(* CODESYS project motor.library
   Company: ESO
   Description: Local Device Control - LDC Motor Library based on State Machine
   Version: 4.2.2.7
   Placeholder: ESO LDC Motor Library
   Author: Dan Popovic
   Title: ESO LDC Motor Library

Project tree, tasks and I/O mapping:
  libraries: Tc2_EtherCAT, * (Beckhoff Automation GmbH); Tc2_IoFunctions, * (Beckhoff Automation GmbH); Tc2_Math, * (Beckhoff Automation GmbH); Tc2_MC2, * (Beckhoff Automation GmbH); Tc2_MC2_Drive, * (Beckhoff Automation GmbH); Tc2_NC, * (Beckhoff Automation GmbH); Tc2_Standard, * (Beckhoff Automation GmbH); Tc2_System, * (Beckhoff Automation GmbH); Tc2_Utilities, * (Beckhoff Automation GmbH); Tc3_EventLogger, * (Beckhoff Automation GmbH); Tc3_Module, * (Beckhoff Automation GmbH); VisuDialogs, * (System); VisuSymbols, 3.5.10.0 (System)
  config/
    Mapping_with_new_EL6688_09_05.xml
    Mapping_with_old_EL6688_03_03.xml
    Mappings_SIM.xml
  00000000-0000-0000-0000-000000000000|config\Mapping_with_new_EL6688_09_05.xml
  00000000-0000-0000-0000-000000000000|config\Mapping_with_old_EL6688_03_03.xml
  00000000-0000-0000-0000-000000000000|config\Mappings_SIM.xml
  doc/
    AM8121_0F20_0000.xti
    EL7041_Phytron_57_500_1.2.xti
    EL7201_9014___AM8121_0F20_0000.xti
    MotorStateMachine.jpg
    Phytron_57_500_1.2_PID.xti
  00000000-0000-0000-0000-000000000000|doc\AM8121_0F20_0000.xti
  00000000-0000-0000-0000-000000000000|doc\EL7041_Phytron_57_500_1.2.xti
  00000000-0000-0000-0000-000000000000|doc\EL7201_9014___AM8121_0F20_0000.xti
  00000000-0000-0000-0000-000000000000|doc\MotorStateMachine.jpg
  00000000-0000-0000-0000-000000000000|doc\Phytron_57_500_1.2_PID.xti
  DUTs/
    Enumerated/
      Common/
        data type E_TIME_MODE
      Motor/
        data type E_DIRECTION
        data type E_MOTOR_AXIS_TYPE
        data type E_MOTOR_COMMAND
        data type E_MOTOR_ERROR
        data type E_MOTOR_EVENT
        data type E_MOTOR_INIT_ACTION
        data type E_MOTOR_INIT_SEQ_STATE
        data type E_MOTOR_INIT_STATE
        data type E_MOTOR_MODE
        data type E_MOTOR_MOVE_TYPE
        data type E_MOTOR_MOVING_STATE
        data type E_MOTOR_POST_INIT_STATE
        data type E_MOTOR_PRE_INIT_STATE
        data type E_MOTOR_RESET_STATE
        data type E_MOTOR_RPC_ERROR
        data type E_MOTOR_STATE
        data type E_MOTOR_STATUS
        data type E_MOTOR_SUBSTATE
        data type E_MOTOR_SWITCH_INDEX
      MultiAxis/
        data type E_MA_ADC_MOUNTING
        data type E_MA_AXES_ID
        data type E_MA_COMMAND
        data type E_MA_EVENT
        data type E_MA_MODE
        data type E_MA_ROTATOR_TYPE
        data type E_MA_RPC_ERROR
        data type E_MA_STATE
        data type E_MA_SUBSTATE
      Tracking/
        data type E_ADC_AXES_ID
        data type E_ADC_MODE
        data type E_DROT_MODE
        data type E_TRK_COMMAND
    Interfaces/
      interface ITrackCtrl: ComputeNextPos, HandleStates, Init, IsError, MoveInPos, MoveInSpeed, Reset
    Structures/
      Astro/
        data type T_ASTRO_ATMOSPHERE
        data type T_ASTRO_EL6688_DATA
        data type T_ASTRO_OUTPUT
        data type T_ASTRO_RA_DEC_RAD
        data type T_ASTRO_STAT
        data type T_ASTRO_TEL_DATA
        data type T_ASTRO_TEL_IF
        data type T_ASTRO_TRACKING_DATA
        data type T_ASTRO_UTC_TIME
        data type T_CPP_DEV_DATA
      CCS_Sim/
        data type T_CCS_CFG
        data type T_CCS_CTRL
        data type T_CCS_STAT
      Common/
        data type T_PTP_TIME
        data type T_TIMEVAL
        data type T_UTC_TIME
      Motor/
        data type T_MOTOR_ACTIVE_LOW
        data type T_MOTOR_AXIS_CFG
        data type T_MOTOR_CFG
        data type T_MOTOR_CTRL
        data type T_MOTOR_INFO
        data type T_MOTOR_INIT_STEP
        data type T_MOTOR_MC_PARAMETER
        data type T_MOTOR_MOTION
        data type T_MOTOR_SIGNAL
        data type T_MOTOR_SPEED
        data type T_MOTOR_STAT
        data type T_MOTOR_SWITCHES
        data type T_POSITION
      MultiAxis/
        data type T_MA_CFG
        data type T_MA_CTRL
        data type T_MA_SM_STAT
        data type T_MA_STAT
        data type T_MA_TOUT_CFG
      Simulation/
        data type T_SIM_MOTOR_CFG
        data type T_SIM_MOTOR_STAT
      Tracking/
        data type T_ADC_CFG
        data type T_ADC_CMD
        data type T_ADC_CTRL
        data type T_ADC_INFO
        data type T_ADC_STAT
        data type T_ADC_UNIT_CFG
        data type T_DROT_CFG
        data type T_DROT_CTRL
        data type T_DROT_INFO
        data type T_DROT_STAT
        data type T_TRK_CFG
        data type T_TRK_CTRL
        data type T_TRK_STAT
  GVLs/
    global variables GVL_TrkDefaultEnvironment
    global variables GVL_TrkSiteConstants
  lib/
  POUs/
    Astro/
      function block FB_ASTRO [ST]: M_Configure, M_CycleUpdate, M_DcAbsoluteTime, M_GetLeapSecond, M_TrkUpdate, M_Update
    CCS/
      function block FB_CCS_SIM [ST]: FB_init, GetParams, RPC_SetCoordinates, SetParams
    Functions/
      function F_astroDms2rad [ST]
      function F_astroHms2rad [ST]
      function F_astroRad2Hms [ST]
      function F_astroSplitHms [ST]
      function F_atan2 [ST]
      function F_DCTIME64_TO_ULINT [ST]
      function F_MOD [ST]
      function F_RAD2DMS_STRING [ST]
      function F_RAD2HMS_STRING [ST]
      function F_slaPa [ST]
      function F_timeGetAbsoluteDcTime [ST]
      function F_timeGetDcTime [ST]
      function F_timeGetUTC [ST]
      function F_timeUTCToJD [ST]
      function F_timeUTCToMJD [ST]
      function F_vltMod [ST]
      function F_vltSign [ST]
    Motor/
      function block FB_MOTOR [ST]: ActionClearNOVRAM, ActionErrExecute, ActionInitAbort, ActionInitComplete, ActionInitExecute, ActionInitReject, ActionMoveExecute, ActionResetExecute, ActionSetPosition, ActionStopExecute, ActionUnexpExecute, ActivityClearingNOVRAM, ActivityInitAborting, ActivityInitializing, ActivityMoving, ActivitySettingPosition, ActivityStopping, CheckForEvents, Dummy_UserExample, M_Configure, M_GetActualPos, M_GetOptimisedDistance, M_GetOptimisedPosition, M_GetRpcErrorText, M_HandleEnabled, M_MotorBrakeControl, M_MotorInitLock, M_MotorInitSeq, M_MotorPostInit, M_MotorPreInit, M_MotorReset, M_NormalizePos, M_NOVRAM_Clear, M_NOVRAM_Load, M_NOVRAM_Save, M_SetError, M_SetRpcStatus, M_UpdateSwitches, RPC_Disable, RPC_Enable, RPC_Init, RPC_MoveAbs, RPC_MoveRel, RPC_MoveVel, RPC_Reset, RPC_SetDebug, RPC_SetLog, RPC_Stop, UserPostInit, UserPostMove, UserPreInit, UserPreMove
      function block FB_MOTOR_BASE [ST]: ActionClearNOVRAM, ActionEnableExecute, ActionErrExecute, ActionInitAbort, ActionInitComplete, ActionInitExecute, ActionInitReject, ActionMoveExecute, ActionResetExecute, ActionSetPosition, ActionStopExecute, ActionUnexpExecute, ActivityClearingNOVRAM, ActivityInitAborting, ActivityInitializing, ActivityMoving, ActivitySettingPosition, ActivityStopping, CheckForEvents, M_GetErrorText, M_GetLogicalState, M_GetTimeInSec, M_LogEventDebug, M_LogEventEnd, M_LogEventError, M_LogEventGeneral, M_LogEventMoveAbs, M_LogEventMoveRel, M_LogEventMoveVel, M_LogEventStart, M_SetStatus, M_SetStatusDescription, ProcessEvents, SetAction, SetEvent, SetState, SetStatus
      function block FB_SIM_MOTOR [ST]: GetLogicalState, RPC_ResetConfig, RPC_SetCouplerState, RPC_SetDelay_Brake, RPC_SetDelay_SwitchActive, RPC_SetDelay_SwitchFind, RPC_SetFailure_BrakeFeedback
    MultiAxis/
      function block FB_MA_ADC [ST]: M_LogCommand, RPC_Disable, RPC_Enable, RPC_Init, RPC_MoveAbs, RPC_MoveAngle, RPC_MoveRel, RPC_MoveVel, RPC_Reset, RPC_StartTrack, RPC_Stop, RPC_StopTrack, User_ComputeAutoPos, User_ComputeNextPos, User_Configure, User_GetParams, User_SetParams
      function block FB_MA_BASE [ST]: ActionDisableExecute, ActionEnableExecute, ActionInitExecute, ActionMoveAbsExecute, ActionMoveVelExecute, ActionResetExecute, ActionStopExecute, ActionTrackExecute, ActivityDisabling, ActivityEnabling, ActivityInitialising, ActivityMoving, ActivityPresetting, ActivityResetting, ActivityStopping, ActivityTracking, CheckForEvents, M_AxesIdle, M_AxesInitialised, M_CheckAxesState, M_CheckError, M_Configure, M_GetMaxPosError, M_GetRpcErrorText, M_HomeMotors, M_LogCommand, M_LogEventGeneral, M_NextMove, M_NextMoveAbs, M_RestartTimer, M_SetInit, M_SetMode, M_SetRpcStatus, M_SetStatus, ProcessEvents, RPC_Init, SetAction, SetEvent, SetState, User_ComputeNextPos, User_Configure, User_GetParams, User_SetParams
      function block FB_MA_DROT [ST]: M_LogCommand, RPC_Disable, RPC_Enable, RPC_Init, RPC_MoveAbs, RPC_MoveAngle, RPC_MoveRel, RPC_MoveVel, RPC_Reset, RPC_StartTrack, RPC_Stop, RPC_StopTrack, User_ComputeNextPos, User_Configure, User_GetParams, User_SetParams
      function block FB_TRK_BASE [ST]: User_Configure, User_GetParams, User_SetParams
    program MAIN [ST]
  Version/
    global variables Global_Version
  VISUs/
    Motor/
      visualisation GUI_Motor001_Cfg
      visualisation GUI_Motor001_Ctrl
      visualisation GUI_Motor002_Cfg
      visualisation GUI_Motor002_Ctrl
    Templates/
      visualisation GUI_TEMPLATE_CCS_SIM
      visualisation GUI_TEMPLATE_MA_ADC
      visualisation GUI_TEMPLATE_MA_DROT
      visualisation GUI_TEMPLATE_MOTOR_CONFIG
      visualisation GUI_TEMPLATE_MOTOR_CONTROL
    Tracking/
      visualisation GUI_ADC_Motor1
      visualisation GUI_ADC_Motor2
      visualisation GUI_CCS_SIM
      visualisation GUI_DROT_Cfg
      visualisation GUI_DROT_Motor
      visualisation GUI_MA_ADC
      visualisation GUI_MA_DROT
  global variables GCL
  text list GlobalTextList
  global variables GPL
*)

// DUTs/Enumerated/Common/E_TIME_MODE
{attribute 'qualified_only'}
{attribute 'strict'}
TYPE E_TIME_MODE :
(
	LOCAL	:= 0,
	UTC		:= 1
);
END_TYPE

// DUTs/Enumerated/Motor/E_DIRECTION
{attribute 'qualified_only'}
{attribute 'strict'}
TYPE E_DIRECTION :
(
	NEGATIVE := 1,
	POSITIVE
);
END_TYPE

// DUTs/Enumerated/Motor/E_MOTOR_AXIS_TYPE
{attribute 'qualified_only'}
{attribute 'strict'}
TYPE E_MOTOR_AXIS_TYPE :
(
	LINEAR				:= 1,
	CIRCULAR,
	CIRCULAR_OPTIMISED
);
END_TYPE

// DUTs/Enumerated/Motor/E_MOTOR_COMMAND
{attribute 'qualified_only'}
{attribute 'strict'}
TYPE E_MOTOR_COMMAND :
(
	NONE	:= 0,
	
	// Commands corresponding to events - MUST match E_MOTOR_EVENT !!!
	RESET,
	INIT,
	STOP,
	ENABLE,
	DISABLE,
	MOTOR_MOVE,
	SET_POSITION,
	CLEAR_NOVRAM
);
END_TYPE

// DUTs/Enumerated/Motor/E_MOTOR_ERROR
{attribute 'qualified_only'}
// 'strict' cannot be used since we mix our own codes with TC codes
//{attribute 'strict'}
TYPE E_MOTOR_ERROR :
(
	OK					:= 0,
	HW_NOT_OP,			
	LOCAL,			
	INIT_ABORTED,		
	TIMEOUT_INIT,
	TIMEOUT_MOVE,
	TIMEOUT_RESET,
	TIMEOUT_SETPOS,
	TIMEOUT_USER_PREINIT,
	TIMEOUT_USER_POSTINIT,
	TIMEOUT_USER_PREMOVE,
	TIMEOUT_USER_POSTMOVE,
	SETPOS,
	STOP,
	
	ABORT,
	SW_LIMIT_LOWER,
	SW_LIMIT_UPPER,
	BRAKE_ACTIVE,
	BRAKE_ENGAGE,
	BRAKE_DISENGAGE,
	SWITCH_NOT_USED,
	ENABLE,
	NOVRAM_READ,
	NOVRAM_WRITE,
	SWITCH_EXIT,
	STOP_LIMITS_BOTH,
	HW_LIMITS_BOTH,
	IN_POS,
	LOCKED,
	SoE_ADS_ERROR,
	SoE_SERCOS_ERROR,

	// Simulator errors
	SIM_NOT_INITIALISED			:= 90,
	SIM_NULL_POINTER			:= 100,	

	// TwinCAT errors
	TC_VEL						:= 16929,	
	TC_NOT_READY_FOR_START		:= 16933,	
	TC_DISABLED_MOVE			:= 16992,	
	TC_BISECTION				:= 17022,	
	TC_MODULO_POS				:= 17026,	
	TC_STOP_ACTIVE				:= 17135,	
	TC_VEL_NEG					:= 17241,	
	TC_TARGET_LSW				:= 17504,	
	TC_TARGET_USW				:= 17505,	
	TC_FOLLOWING_ERROR			:= 17744,	
	TC_NOT_READY				:= 18000,	
	TC_IN_POS_6_SEC				:= 19207	

);
END_TYPE

// DUTs/Enumerated/Motor/E_MOTOR_EVENT
{attribute 'qualified_only'}
{attribute 'strict'}
TYPE E_MOTOR_EVENT :
(
	NONE	:= 0,
	
	(* events corresponding to commands - MUST match E_MOTOR_COMMAND *)
	RESET,
	INIT,
	STOP,
	ENABLE,
	DISABLE,
	MOTOR_MOVE,
	SET_POSITION,
	CLEAR_NOVRAM,
	
	(* 
		Events corresponding to internal events 
	*)
	
	MOVEDONE,		// Needed for detection of HW failures during initialisation
	STOPDONE,
	ENABLEDONE,
	DISABLEDONE,
	INITDONE,
	SETPOSDONE,
	

	HWOK,
	ERRLOCAL,
	ERRHW,
	ERRRESET,
	ERRFAULT,
	ERRINIT,
	ERRSTOP,
	ERRENABLE,
	ERRDISABLE,
	ERRBRAKE,
	ERRINPOS,
	ERRLOCKED,
	ERRTARGETPAR,
	ERRUSERPREINIT,
	ERRUSERPREMOVE,
	ERRUSERPOSTINIT,
	ERRUSERPOSTMOVE,
	TIMEOUT_MOVE,
	TIMEOUT_SETPOS,
	SW_LIMIT_LOWER,
	SW_LIMIT_UPPER
	
);
END_TYPE

// DUTs/Enumerated/Motor/E_MOTOR_INIT_ACTION
TYPE E_MOTOR_INIT_ACTION :
(
	MOTOR_INIT_ACTION_END				:= 0,
	MOTOR_INIT_ACTION_FIND_INDEX,
	MOTOR_INIT_ACTION_FIND_REF_LE,
	MOTOR_INIT_ACTION_FIND_REF_UE,
	MOTOR_INIT_ACTION_FIND_LHW,
	MOTOR_INIT_ACTION_FIND_UHW,
	MOTOR_INIT_ACTION_DELAY,
	MOTOR_INIT_ACTION_MOVE_ABS,
	MOTOR_INIT_ACTION_MOVE_REL,
	MOTOR_INIT_ACTION_CALIB_ABS,
	MOTOR_INIT_ACTION_CALIB_REL,
	MOTOR_INIT_ACTION_CALIB_SWITCH,
	// The following steps cannot be configured in the INIT sequence
	MOTOR_INIT_ACTION_STEP1_START,
	MOTOR_INIT_ACTION_STEP1_EXECUTE,
	MOTOR_INIT_ACTION_STEP2_START,
	MOTOR_INIT_ACTION_STEP2_EXECUTE,
	MOTOR_INIT_ACTION_STOP
);
END_TYPE

// DUTs/Enumerated/Motor/E_MOTOR_INIT_SEQ_STATE
TYPE E_MOTOR_INIT_SEQ_STATE :
(
	MOTOR_INIT_SEQ_STATE_START				:= 0,
	MOTOR_INIT_SEQ_STATE_EXECUTE,
	MOTOR_INIT_SEQ_STATE_END
);
END_TYPE

// DUTs/Enumerated/Motor/E_MOTOR_INIT_STATE
TYPE E_MOTOR_INIT_STATE :
(
	MOTOR_INIT_STATE_START				:= 0,
	MOTOR_INIT_STATE_RESET,
	MOTOR_INIT_STATE_WAIT_READY,
	MOTOR_INIT_STATE_PRE_INIT,
	MOTOR_INIT_STATE_USER_PRE_INIT,
	MOTOR_INIT_STATE_INIT_SEQ,
	MOTOR_INIT_STATE_INIT_LOCK,
	MOTOR_INIT_STATE_POST_INIT,
	MOTOR_INIT_STATE_USER_POST_INIT,
	MOTOR_INIT_STATE_SAVE_NOVRAM,
	MOTOR_INIT_STATE_END
);
END_TYPE

// DUTs/Enumerated/Motor/E_MOTOR_MODE
{attribute 'qualified_only'}
{attribute 'strict'}
TYPE E_MOTOR_MODE :
(
	POS				:= 0,
	VEL
);
END_TYPE

// DUTs/Enumerated/Motor/E_MOTOR_MOVE_TYPE
{attribute 'qualified_only'}
{attribute 'strict'}
TYPE E_MOTOR_MOVE_TYPE :
(
	NONE	:= 0,
	
	ABSOLUTE,
	RELATIVE,
	VELOCITY,
	TRACKING

);
END_TYPE

// DUTs/Enumerated/Motor/E_MOTOR_MOVING_STATE
TYPE E_MOTOR_MOVING_STATE :
(
	MOTOR_MOVING_STATE_NONE	:= 0,
	MOTOR_MOVING_STATE_ENABLE,
	MOTOR_MOVING_STATE_WAIT_BRAKES,
	MOTOR_MOVING_STATE_USER_PRE_MOVE,
	MOTOR_MOVING_STATE_WAIT_ABSOLUTE,
	MOTOR_MOVING_STATE_WAIT_OPTIMISED,
	MOTOR_MOVING_STATE_WAIT_VELOCITY,
	MOTOR_MOVING_STATE_USER_POST_MOVE,
	MOTOR_MOVING_STATE_APPLY_BRAKES,
	MOTOR_MOVING_STATE_DISABLE,
	MOTOR_MOVING_STATE_CHECK_IN_POS,
	MOTOR_MOVING_STATE_END
);
END_TYPE

// DUTs/Enumerated/Motor/E_MOTOR_POST_INIT_STATE
TYPE E_MOTOR_POST_INIT_STATE :
(
	MOTOR_POST_INIT_STATE_START	:= 0,
	MOTOR_POST_INIT_STATE_WRITE,
	MOTOR_POST_INIT_STATE_END
);
END_TYPE

// DUTs/Enumerated/Motor/E_MOTOR_PRE_INIT_STATE
TYPE E_MOTOR_PRE_INIT_STATE :
(
	MOTOR_PRE_INIT_STATE_START	:= 0,
	MOTOR_PRE_INIT_STATE_READ,
	MOTOR_PRE_INIT_STATE_GET_USER_UNITS,
	MOTOR_PRE_INIT_STATE_WRITE,
	MOTOR_PRE_INIT_STATE_END
);
END_TYPE

// DUTs/Enumerated/Motor/E_MOTOR_RESET_STATE
TYPE E_MOTOR_RESET_STATE :
(
	MOTOR_RESET_STATE_START	:= 0,
	MOTOR_RESET_STATE_SoE_RESET,
	MOTOR_RESET_STATE_SoE_WAIT_RESET,
	MOTOR_RESET_STATE_RESET_AXIS,
	MOTOR_RESET_STATE_WAIT,
	MOTOR_RESET_STATE_END
);
END_TYPE

// DUTs/Enumerated/Motor/E_MOTOR_RPC_ERROR
{attribute 'qualified_only'}
{attribute 'strict'}
TYPE E_MOTOR_RPC_ERROR :
(
	OK						:= 0,
	NOT_OP					:= -1,			
	NOT_NOTOP_READY			:= -2,			
	NOT_NOTOP_NOTREADY		:= -3,			
	LOCAL					:= -4,			
	SW_LIMIT_LOWER			:= -5,			
	SW_LIMIT_UPPER			:= -6,			
	INIT_WHILE_MOVING		:= -7,
	VEL_ZERO				:= -8,			
	VEL_NEG					:= -9,			
	VEL_MAX					:= -10			
);
END_TYPE

// DUTs/Enumerated/Motor/E_MOTOR_STATE
{attribute 'qualified_only'}
{attribute 'strict'}
TYPE E_MOTOR_STATE :
(
	NONE	:= 0,
	NOTOP,
	OP
);
END_TYPE

// DUTs/Enumerated/Motor/E_MOTOR_STATUS
{attribute 'qualified_only'}
{attribute 'strict'}
TYPE E_MOTOR_STATUS :
(
	OK	:= 0,
	ERROR,
	
	STANDING,
	MOVING

);
END_TYPE

// DUTs/Enumerated/Motor/E_MOTOR_SUBSTATE
{attribute 'qualified_only'}
{attribute 'strict'}
TYPE E_MOTOR_SUBSTATE :
(
	NONE					:= 0,
	
	NOTOP_NOTREADY			:= 100,
	NOTOP_READY				:= 101,
	NOTOP_INITIALIZING		:= 102,
	NOTOP_ABORTING			:= 107,
	NOTOP_CLEARING_NOVRAM	:= 108,
	
	NOTOP_ERROR				:= 199,
	
	
	OP_STANDSTILL			:= 216,            
	OP_MOVING				:= 217,
	OP_SETTING_POS			:= 218,
	OP_STOPPING				:= 219,
	
	OP_ERROR				:= 299
);
END_TYPE

// DUTs/Enumerated/Motor/E_MOTOR_SWITCH_INDEX
{attribute 'qualified_only'}
{attribute 'strict'}
TYPE E_MOTOR_SWITCH_INDEX :
(
	LSTOP	:= 0,
	LHW		:= 1,
	REF		:= 2,
	INDEX	:= 3,
	UHW		:= 4,
	USTOP	:= 5
);
END_TYPE

// DUTs/Enumerated/MultiAxis/E_MA_ADC_MOUNTING
TYPE E_MA_ADC_MOUNTING :
(
	// ADC positions should be the same due to oposite mounting of ADC units,
	// i.e. ADC2 = ADC1
	MA_ADC_MOUNTING_OPOSITE_SIDE := 0,
	// ADC positions should have oposite vales due to the same mounting of both ADC units,
	// i.e. ADC2 = -ADC1
	MA_ADC_MOUNTING_SAME_SIDE := 1
);
END_TYPE

// DUTs/Enumerated/MultiAxis/E_MA_AXES_ID
{attribute 'qualified_only'}
{attribute 'strict'}
TYPE E_MA_AXES_ID :
(
	ALL_AXES := 0,
	AXIS_1,
	AXIS_2,
	AXIS_3,
	AXIS_4,
	AXIS_5,
	AXIS_6
);
END_TYPE

// DUTs/Enumerated/MultiAxis/E_MA_COMMAND
{attribute 'qualified_only'}
{attribute 'strict'}
TYPE E_MA_COMMAND :
(
	NONE	:= 0,
	
	// Commands corresponding to events - MUST match E_MA_EVENT !!!
	RESET,
	INIT,
	STOP,
	ENABLE,
	DISABLE,
	MA_MOVE,
	START_TRACK,
	STOP_TRACK
);
END_TYPE

// DUTs/Enumerated/MultiAxis/E_MA_EVENT
{attribute 'qualified_only'}
{attribute 'strict'}
TYPE E_MA_EVENT :
(
	NONE	:= 0,
	
	(* events corresponding to commands - MUST match E_MA_COMMAND *)
	RESET,
	INIT,
	STOP,
	ENABLE,
	DISABLE,
	MA_MOVE,
	START_TRACK,
	STOP_TRACK,
	
	(* 
		Events corresponding to internal events 
	*)
	
	MOVEDONE,		// Needed for detection of HW failures during initialisation
	STOPDONE,
	ENABLEDONE,
	DISABLEDONE,
	INITDONE,
	TRACKDONE,
	TRACKEXIT,		// EICSSW-706: Tracking error >=  cfg.lrTrkThreshold => PRESETTING
	PRESETDONE,		// EICSSW-706: Presetting error < cfg.lrTrkThreshold => TRACKING
	

	HWOK,
	ERRLOCAL,
	ERRHW
	
);
END_TYPE

// DUTs/Enumerated/MultiAxis/E_MA_MODE
TYPE E_MA_MODE :
(
	// WARNING: modes shall be a positive number
	MA_MODE_ENG	:= 0
);
END_TYPE

// DUTs/Enumerated/MultiAxis/E_MA_ROTATOR_TYPE
{attribute 'qualified_only'}
{attribute 'strict'}
TYPE E_MA_ROTATOR_TYPE :
(
	DROT 	:= 0,	// Derotator
	ADAPTER := 1,	// Adapter
	ROTATOR := 2	// Rotator
);
END_TYPE

// DUTs/Enumerated/MultiAxis/E_MA_RPC_ERROR
{attribute 'qualified_only'}
{attribute 'strict'}
TYPE E_MA_RPC_ERROR :
(
	OK						:=  0,
	NOT_OP					:= -1,			
	NOT_NOTOP_READY	    	:= -2,			
	NOT_NOTOP_NOTREADY		:= -3,			
	LOCAL					:= -4,			
	SW_LIMIT_LOWER			:= -5,			
	SW_LIMIT_UPPER			:= -6,			
	INIT_WHILE_MOVING		:= -7,
	VEL_ZERO				:= -8,			
	VEL_NEG					:= -9,			
	VEL_MAX					:= -10			
);
END_TYPE

// DUTs/Enumerated/MultiAxis/E_MA_STATE
{attribute 'qualified_only'}
//{attribute 'strict'}
TYPE E_MA_STATE :
(
	NONE	:= 0,
	NOTOP,
	OP
);
END_TYPE

// DUTs/Enumerated/MultiAxis/E_MA_SUBSTATE
{attribute 'qualified_only'}
//{attribute 'strict'}
TYPE E_MA_SUBSTATE :
(
	NONE				:=   0,
	
	NOTOP_NOTREADY		:= 100,
	NOTOP_READY			:= 101,
	NOTOP_INITIALISING	:= 102,
	NOTOP_ABORTING		:= 107,
	
	NOTOP_RESETTING		:= 109,
	NOTOP_ENABLING		:= 110,

	NOTOP_ERROR			:= 199,

	
	OP_DISABLING 		:= 205,
	OP_STANDSTILL		:= 216,            
	OP_MOVING			:= 217,
	OP_SETTING_POS		:= 218,
	OP_STOPPING			:= 219,
	OP_TRACKING			:= 220,
	OP_PRESETTING		:= 221,

	OP_ERROR			:= 299

);
END_TYPE

// DUTs/Enumerated/Tracking/E_ADC_AXES_ID
{attribute 'qualified_only'}
{attribute 'strict'}
TYPE E_ADC_AXES_ID :
(
	ALL_AXES := 0,
	ADC_1,
	ADC_2
);
END_TYPE

// DUTs/Enumerated/Tracking/E_ADC_MODE
{attribute 'qualified_only'}
{attribute 'strict'}
TYPE E_ADC_MODE :
(
	// WARNING: modes shall be a positive number
	ENG   := 0, 
	OFF   := 1,
	AUTO  := 2
);
END_TYPE

// DUTs/Enumerated/Tracking/E_DROT_MODE
{attribute 'qualified_only'}
{attribute 'strict'}
TYPE E_DROT_MODE :
(
	ENG		:= 0,
	STAT	:= 1,
	SKY		:= 2,
	ELEV	:= 3,
	USER	:= 4
);
END_TYPE

// DUTs/Enumerated/Tracking/E_TRK_COMMAND
{attribute 'qualified_only'}
{attribute 'strict'}
TYPE E_TRK_COMMAND :
(
	NONE			:= 0,
	INIT			:= 1,
	STOP, 
	TRK_MOVE,
	START_TRACK,
	STOP_TRACK,
	RESET,
	ENABLE,
	DISABLE,
	MOVE_MASTER
);
END_TYPE

// DUTs/Structures/Astro/T_ASTRO_ATMOSPHERE
// Structure containing atmospheric conditions.
// To be updated by the WS driver, i.e. "scanning" from TEL
TYPE T_ASTRO_ATMOSPHERE :
STRUCT
	lrTemperature:	LREAL   := 12.0;	// Air temperature [degC]
	lrPressure:		LREAL   := 743.0;	// Atmospheric Pressure [mbar]
	lrHumidity:		LREAL   := 0.2;		// Relative humidity [0.0..1.0]
END_STRUCT
END_TYPE

// DUTs/Structures/Astro/T_ASTRO_EL6688_DATA
TYPE T_ASTRO_EL6688_DATA :
STRUCT
	Control_value_update_toggle:	BOOL;
	External_device_not_connected:	BOOL;
	Internal_time_stamp:			ULINT;
	External_time_stamp:			ULINT;
END_STRUCT
END_TYPE

// DUTs/Structures/Astro/T_ASTRO_OUTPUT
TYPE T_ASTRO_OUTPUT :
STRUCT
	stCoordinates:		T_ASTRO_TEL_DATA;
	stAtmosphere:		T_ASTRO_ATMOSPHERE;
	stUtcTime:			T_ASTRO_UTC_TIME;
	stTrackingData:		T_ASTRO_TRACKING_DATA;		// TODO: Only for system without C++ module
END_STRUCT
END_TYPE

// DUTs/Structures/Astro/T_ASTRO_RA_DEC_RAD
// Structure to be updated by the WS driver, i.e. "scanning" from TEL
TYPE T_ASTRO_RA_DEC_RAD :
STRUCT
	ra:       		LREAL;				// RA  [rad]
	dec: 			LREAL;				// Dec [rad]
END_STRUCT
END_TYPE

// DUTs/Structures/Astro/T_ASTRO_STAT
TYPE T_ASTRO_STAT :
STRUCT
	bInitialised:	BOOL	:= FALSE;
	bConfigured:	BOOL 	:= FALSE;	// If TRUE, FB has been configured
	bBadTimeSignal: BOOL 	:= TRUE;

	// Parameters for reading the Leap Second from EL6688
	sAmsNetId: 			T_AmsNetId	:= '';
	nAmsPort: 			T_AmsPort	:= 0;

	bGetLeapSecond:		BOOL 		:= FALSE;	// Trigger for Leap Second SDO read
	bLeapSecondRead:	BOOL 		:= FALSE;	// If TRUE, Leap Second SDO has been read

	mode:     		DINT;
	nLeapSecond:	DINT;

	tDcTime:		ULINT;			// T_ULARGE_INTEGER;
	tUtcTime:		ULINT;			// T_ULARGE_INTEGER;

	sDcTime:		STRING(32);		// System DC time as string
	sUtcTime:		STRING(32);		// UTC time as string

	(* Error handling status *)
	nErrorCode: 	DINT 	:= 0;	(* TODO Error code *)
	nStatus: 		DINT	:= 0; 	(* TODO status *)

	sErrorText: 	STRING 	:= 'NOT INITIALISED';	(* Error description, e.g. 'OK', 'WRONG TIME', etc *)
	sStatus: 		STRING 	:= 'OK';				(* Status in textual form, e.g. 'ACTIVE' *)

	nCounter:		UDINT	:= 0;								(* Alive counter *)
END_STRUCT
END_TYPE

// DUTs/Structures/Astro/T_ASTRO_TEL_DATA
// Structure to be updated by the WS driver, i.e. "scanning" from TEL
TYPE T_ASTRO_TEL_DATA :
STRUCT
	ra_hms:     	LREAL;				// RA  [hms]
	dec_dms: 		LREAL;				// Dec [dms]

	equinox: 		LREAL	:= 2000.0;
	latitude:		LREAL;				// TEL latitude  [rad]
	longitude:		LREAL;				// TEL longitude [rad]

	adaPos_deg: 	LREAL	:= 0.0;		// TODO: Adapter position [deg]
	corrPos_deg: 	LREAL	:= 0.0;		// TODO: Corrector position [deg]
END_STRUCT
END_TYPE

// DUTs/Structures/Astro/T_ASTRO_TEL_IF
// Structure to be updated by the WS driver, i.e. "scanning" from TEL.
// Normally, this will by done via OPC UA.
TYPE T_ASTRO_TEL_IF :
STRUCT
	equinox: 		LREAL	:= 2000.0;
	latitude:		LREAL	:= GCL.C_LATITUDE_ELT;	// TEL latitude  [rad]
	longitude:		LREAL	:= GCL.C_LONGITUDE_ELT;	// TEL longitude [rad]

	ra_hms:       	LREAL;							// TODO: RA  [hhmmss.ttt ?] 
	dec_dms: 		LREAL;							// TODO: Dec [ddmmss.ttt ?]
	
	lrTemperature:	LREAL   := 12.0;				// Air temperature [degC]
	lrPressure:		LREAL   := 743.0;				// Atmospheric Pressure [mbar]
	lrHumidity:		LREAL   := 0.2;					// Relative humidity [0.0..1.0]

	adaPos_deg: 	LREAL	:= 0.0;					// TODO: Adapter position [deg]
	corrPos_deg: 	LREAL	:= 0.0;					// TODO: Corrector position [deg]
END_STRUCT
END_TYPE

// DUTs/Structures/Astro/T_ASTRO_TRACKING_DATA
TYPE T_ASTRO_TRACKING_DATA :
STRUCT
	// TODO: Specify units in the coment.
	//		Should pa be pa_r, etc?
	gmst    : LREAL;	// Greenwich Mean Sidereal Time
	pa      : LREAL;	// parallactic angle [rad]
	pa_deg  : LREAL;	// parallactic angle [deg]
	alt     : LREAL;	// altitude [rad]
	alt_deg : LREAL;	// altitude [deg]
	ha      : LREAL;	// hour angle [rad]
	az      : LREAL;	// azimuth [rad]
	az_deg  : LREAL;	// azimuth [deg]
	ra_r    : LREAL;	// RA  [rad]
	dec_r   : LREAL;	// Dec [rad]
	// TODO: New 
	ra_hms  : LREAL;	// RA  [Hms]
	dec_dms : LREAL;	// Dec [Dms]
	ha_hms  : LREAL;	// hour angle [Hms]
	ha_deg  : LREAL;	// hour angle [deg]
	fr   	: LREAL;	// Field rotation [rad]
	pr		: LREAL;	// Pupil rotation [rad]
END_STRUCT
END_TYPE

// DUTs/Structures/Astro/T_ASTRO_UTC_TIME
TYPE T_ASTRO_UTC_TIME :
STRUCT
	dcTime:   			ULINT;
	mode:     			DINT;
	nLeapSecond:		DINT;
	bLeapSecondQuality:	BOOL;	// If TRUE, Leap Second is successfully read
	bBadTimeSignal: 	BOOL := TRUE;
END_STRUCT
END_TYPE

// DUTs/Structures/Astro/T_CPP_DEV_DATA
// Output structure generated by the C++ coordinate transformation module.
// It contains complete info about TEL position, atmospheric conditions and
// DC System time and UTC time.
// The structure should be mapped/linked to tracking device input. 
TYPE T_CPP_DEV_DATA :
STRUCT
	stCoordinates:	T_ASTRO_TEL_DATA;
	stAtmosphere:	T_ASTRO_ATMOSPHERE;
	stUtcTime:		T_ASTRO_UTC_TIME;
	stTrackingData:	T_ASTRO_TRACKING_DATA;
END_STRUCT
END_TYPE

// DUTs/Structures/CCS_Sim/T_CCS_CFG
TYPE T_CCS_CFG:
STRUCT
	site:     TrkSiteConstants;
END_STRUCT
END_TYPE

// DUTs/Structures/CCS_Sim/T_CCS_CTRL
TYPE T_CCS_CTRL:
STRUCT
	meanCoordinates: TrkMeanCoordinates;
	environment:     TrkEnvironment;
	motion:          TrkPolarMotion;
	wavelength:      LREAL := 600;
	dut:             LREAL := 0.0;
	equinox:         LREAL := 2000.0;
END_STRUCT
END_TYPE

// DUTs/Structures/CCS_Sim/T_CCS_STAT
TYPE T_CCS_STAT:
STRUCT
	apparent   :        TrkApparentCoordinates;
	observed   :        TrkObservedCoordinates;
	environment:        TrkEnvironment;
	data       :        TrkComputation;
	nTimeMode  :        DINT := 0;
	sTimeMode  :        STRING := '';
	sDcTime    :        STRING := '';
	lDcTime    :        LINT := 0;
END_STRUCT
END_TYPE

// DUTs/Structures/Common/T_PTP_TIME
(*
typedef struct _PTPTime
{
	ULONGLONG internal;
	ULONGLONG external;
	bool not_connected;
	bool update_toggle;
	LONGLONG dcTcOffset;
} PTPTime, *PPTPTime;
*)
TYPE T_PTP_TIME :
STRUCT
END_STRUCT
END_TYPE

// DUTs/Structures/Common/T_TIMEVAL
TYPE T_TIMEVAL :
STRUCT
    tv_sec:		UDINT;	// seconds since midnight January 1,1970 UTC
    tv_usec:	DINT;  	// and microseconds
END_STRUCT
END_TYPE

// DUTs/Structures/Common/T_UTC_TIME
TYPE T_UTC_TIME :
STRUCT
	dcTime:   ULINT;
	mode:     DINT;
END_STRUCT
END_TYPE

// DUTs/Structures/Motor/T_MOTOR_ACTIVE_LOW
TYPE T_MOTOR_ACTIVE_LOW :
STRUCT
	bValue:	BOOL	:= FALSE;
END_STRUCT
END_TYPE

// DUTs/Structures/Motor/T_MOTOR_AXIS_CFG
TYPE T_MOTOR_AXIS_CFG :
STRUCT
	////////////////////////////////////////////////////////////////////////
	// The following configuration parameters are read from Axis on INIT. //
	////////////////////////////////////////////////////////////////////////
	
	lrScaleFactor:	LREAL 	:= 1.0;				// Read from Axis on INIT
	lrModuloFactor: LREAL 	:= 360.0;			// Read from Axis on INIT
	lrAccel: 		LREAL 	:= 30.0;			// Read from Axis on INIT
	lrDecel: 		LREAL 	:= 30.0;			// Read from Axis on INIT
	lrJerk: 		LREAL 	:= 100;				// Read from Axis on INIT
	lrMaxVelocity:	LREAL 	:= 0.001;			// Read from Axis on INIT
	lrMaxPosLag:	LREAL 	:= 0.0;				// Read from Axis on INIT
	sUnits:			STRING(16) 	:= 'UNKNOWN';	// Read from Axis on INIT using ADS

END_STRUCT
END_TYPE

// DUTs/Structures/Motor/T_MOTOR_CFG
TYPE T_MOTOR_CFG :
STRUCT
	//////////////////////////////////////////////////////////
	// Parameters configurable from WS, Cfg GUI or directly //
	//////////////////////////////////////////////////////////
	
	// Backlash compensation value [UU], direction given by the sign, 
	// 0:	no backlash compensation, 
	// >0:	approach from positive direction, 
	// <0:	approach from negative direction
	lrBacklash:			LREAL 	:= 0.0;		
	lrDefaultVelocity:	LREAL 	:= 0.01;	// Default velocity for position mode [UU]

	// SW Limits.
	// If both limits are set to zero, limits are not used.
	lrMaxPosition:		LREAL 	:= 0.0;	//  [UU]
	lrMinPosition:		LREAL 	:= 0.0;	//  [UU]

	nAxisType:			DINT	:= E_MOTOR_AXIS_TYPE.LINEAR;

	// Timeouts
	nTimeoutInit:		DINT 	:= 60000;	(* Timeout for complete INIT sequence [ms] *)
	nTimeoutMove:		DINT 	:= 60000;	(* Timeout for a single move [ms] *)
	nTimeoutSwitch:		DINT 	:= 15000;	(* Timeout for exiting a switch [ms] *)


	// Brake handling
	bUseBrake:			BOOL	:= FALSE;
	bActiveLowBrake:	BOOL	:= FALSE;

	// ActiveLow configuration for switches. Default is 'FALSE'. 
	bArrActiveLow:		ARRAY [E_MOTOR_SWITCH_INDEX.LSTOP..E_MOTOR_SWITCH_INDEX.USTOP] OF T_MOTOR_ACTIVE_LOW;
	
	// ActiveLow configuration for in-position switch. Default is 'FALSE'. 
	bActiveLowInPos:	BOOL	:= FALSE;

	// Default INIT sequence - Just calibrate to zero.
	strArrInitSeq:		ARRAY [1..10] OF T_MOTOR_INIT_STEP := [
											(nAction:=9, lrValue1:=0.0, lrValue2:=0.0),
											(nAction:=0, lrValue1:=0.0, lrValue2:=0.0),
											(nAction:=0, lrValue1:=0.0, lrValue2:=0.0),
											(nAction:=0, lrValue1:=0.0, lrValue2:=0.0),
											(nAction:=0, lrValue1:=0.0, lrValue2:=0.0),
											(nAction:=0, lrValue1:=0.0, lrValue2:=0.0),
											(nAction:=0, lrValue1:=0.0, lrValue2:=0.0),
											(nAction:=0, lrValue1:=0.0, lrValue2:=0.0),
											(nAction:=0, lrValue1:=0.0, lrValue2:=0.0),
											(nAction:=0, lrValue1:=0.0, lrValue2:=0.0)];
											
	// Function lock
	bLock:			BOOL	:= FALSE;	// If TRUE, motor is locked
	lrLockPos:		LREAL 	:= 0.0;		// Locked position [UU]
	lrLockTol:		LREAL 	:= 0.0;		// Tolerance for in-locked position [UU]
	
	// User defined methods execution
	bExecUserPreInit:	BOOL	:= FALSE;
	bExecUserPostInit:	BOOL	:= FALSE;
	bExecUserPreMove:	BOOL	:= FALSE;
	bExecUserPostMove:	BOOL	:= FALSE;
	
	// Misc checks
	bCheckInPos:		BOOL	:= FALSE;	// If TRUE, check if i_bInPos signal is active after move
	bDisableAfterMove:	BOOL	:= FALSE;	// If TRUE, disable motor after each move
	
	// SoE drives (Sercos over EtherCAT) , e.g. AX5000, need special Reset procedure FB_SoEReset()
	// in case of drive failure.
	// Other drives, i.e. CoE drives (Can over EtherCAT), are reset with the standard MC_Reset().
	// IMPORTANT NOTE: For the AX5000 the "Wait For WcState is OK" flag 
	//                 has to be activated in the Advanced EtherCAT Settings/General/Behavior.
	bSoE_Drive:			BOOL	:= FALSE;	// If TRUE, SoE drive, e.g. AX5000), default CoE, i.e. FALSE

	// Logging
	bLogExtTime:		BOOL 	:= FALSE;		// If TRUE, use external time in event logs. Default FALS
	bDebug:				BOOL 	:= FALSE;		// If TRUE, show event logs of Debug type. Default FALSE.
	bLog:				BOOL 	:= TRUE;		// If TRUE, log events. Default TRUE.
	
END_STRUCT
END_TYPE

// DUTs/Structures/Motor/T_MOTOR_CTRL
TYPE T_MOTOR_CTRL :
STRUCT
	// Command value and execution flag
	nCommand:	E_MOTOR_COMMAND	:= E_MOTOR_COMMAND.NONE;// See E_MOTOR_COMMAND 
	bExecute:	BOOL;									// Triggers command execution
	
	// If bLocalCmd is TRUE, commands are accepted in Local mode.
	// This var is set by each button press in local GUI.
	// This var is reset after each command handling.
	// Each button in local GUI has to have the first command:
	//    m_Instance.ctrl.bLocalCmd := TRUE;
	// This variable is not available in OPC UA namespace.
	//
	{attribute 'OPC.UA.DA' := '0'}
	bLocalCmd:		BOOL	:= FALSE;				

	// Motion parameters
	nMoveType:		DINT	:= E_MOTOR_MOVE_TYPE.NONE;
	nDirection:		DINT 	:= MC_Positive_Direction;
	lrPosition: 	LREAL 	:= 0.0;		// Value for MOVE_ABS
	lrOffset: 		LREAL 	:= 0.0;		// Value for MOVE_REL (EICSSW-781)
	lrVelocity:		LREAL 	:= 0.0001;

END_STRUCT
END_TYPE

// DUTs/Structures/Motor/T_MOTOR_INFO
TYPE T_MOTOR_INFO :
STRUCT
(*
Driver Information 

Change Log:
	0.1	2016-07-14	- Snapshot - Porting from FB_MOTOR_CONTROL.
		2016-07-14	- Snapshot - MC_Halt instead of MC_Stop.
					- Implemented NOVRAM Load/Save - to be tested.
					- Signals monitored during STOPPING in INIT.
					- Removed most of Lamp code (this was the starting point)
		2016-08-09	- Implemented NOVRAM R/W.
					- Both limit switches check done only after NOVRAM is loaded.
					- Created first Motor.library.
	0.2 2017-01-30	- Simulator FB_SIM_MOTOR improvements ONLY.
					- Addition of simulator status structure.
					- Improved recognition of INIT command.
					- Fixed handling of REF_LE signal level.
					- Addition of RPC calls.
	0.3 2017-06-23	- WARNING: Compatible with TC 3.1.4020 or later.
					- Addition of Simulator handling of STOP signals.
					- Additional checks for Move Done, i.e. CommandAborted and NotMoving.
					- Addition of method M_GetActualPos().
					- Normalise set position for circular-optimised.
					- Additional checks for STOP switches.
	0.4 2017-08-11	- Improved stopping using fbHalt().
					- STOP timeout increased from 3 to 10 sec.
					- Handling of E_MOTOR_EVENT.ERRSTOP while Stopping.
					- Direction disabled depending on L/U STOP active level - no relaxed case for INIT.
					- Addition of State Machine GUI.
	0.5 2017-08-31	- Big cleanup.
					- Removed unused cfg variables lrTolerance and lrToleranceEnc.
					- Removed unused cfg variable cfg.lrScaleFactor.
					- Renamed cfg.nTypeAxis to cfg.nAxisType.
					- Corrected stopping while searching for switches.
					- Renamed bActiveLow to bValue in T_MOTOR_ACTIVE_LOW. 
					- Removed stat.lrInPosTolerance.
					- Renamed stat.bLimSwitch* to stat.bStopSwitch*.
					- Removed E_MOTOR_HW_STATUS.
	0.6 2017-09-01	- Motor stopped on timeout in Position mode.
					- Removed substate E_MOTOR_SUBSTATE.OP_DISABLING.
	0.7 2017-09-07	- Completed RPC Calls.
	0.8 2017-10-06	- Addition of ctrl.bLocalCmd.
					- Addition of m_Instance.ctrl.bLocalCmd := TRUE; to each GUI button.
					- Addition of stat.nCounter 'alive' counter.
					- Addition of E_MOTOR_EVENT.ERRLOCAL.
					- Added check for stat.bLocal in RPC Calls.
					- Removed RPC_SetPos.
	0.9 2017-10-12	- Replaced nInternalEvent to nEvent in Activities.
					- Implemented handling of hitting SW limits.
					- Improved failure handling during INIT.
	0.10 2018-01-24	- Handling of Locked mode.
					- Addition of 'i_bInPos	AT %I*:	BOOL' signal for in-position check
					- Addition of config parameters for User Methods.
					- Addition of UserPreInit() and UserPostInit() methods.
					- Addition of UserPreMove() and UserPostMove() methods.
					- Added calls to UserPreInit() and UserPostInit() methods in ActivityInitializing().
					- Added calls to UserPreMove() and UserPostMove() methods in ActivityMoving().
					- Additonal configuration parameters in Config GUI.
					- Changed nCmdCycleCounter type from DINT to UDINT.
					- Implemented FB_MOTOR::M_NOVRAM_Clear().
					- Corrected handling of E_MOTOR_EVENT.STOP in E_MOTOR_SUBSTATE.NOTOP_*.
					- Implemented Auto Disable.
					- Implemented In-Position check
	0.11 2018-01-25	- Completed handling of Locked mode.
	0.12 2018-01-30	- If configured for Disable After Move, axis disabled after INIT.
					- Additions of ENABLE/DISABLE AXIS buttons.
	0.13 2018-02-02	- Addition of MOTOR_INIT_STATE_WAIT_READY state to wait for AxisReady after Reset.
	1.3.0.0			- Moved nCmdCycleCounter to T_MOTOR_STAT.
					- Addition of {attribute 'OPC.UA.DA' := '0'} to block unwanted FB's and vars.
					- Addition of {attribute 'OPC.UA.DA' := '0'} for all VAR_INST.
	1.4.0.0			- RPC calls return INT.
					- Addition of E_MOTOR_RPC_ERROR.
	1.5.0.0			- Renaming of methods - prefix M_.
					- Addition of M_GetErrorText() and M_SetStatusDescription().
					- Axis User Units read with ADSREAD.
					- Improved State Machine.
					- Addition of sLibVersion.
	1.7.0.0			- Check for SW Limits in RPC_MoveAbs() and RPC_MoveRel().
	1.8.0.0			- Added support for SoE Drives Reset.
	1.8.0.1			- Added stat.nCycleTime.
					- Added one cycle time to UTC coming from ASTRO.
	2.0.0.0			- Code grouped in subdirectories.
	2.1.0.0			- If not OP, motor goes to NOTOP_FAILURE.
					- Corrected simulator handling of CouplerStatus.
	2.2.0.0			- axisCfg structure moved to stat.axis.
					- Addition of stat.axis.lrMaxPosLag.
					- In case of both STOP or HW limits being active, motor goes to NOTOP_ERROR.
	2.3.0.0			- Going back to TC3.1.4022.14 due to increased library size.
					- Renaming States STANDBY->NOTOP & FAILURE->ERROR.
	3.0.0.0			- WARNING: Requires TwinCAT 3.1 build 4022.20 or higher.
					- Projects need Tc3_EventLogger library included in References.
					- Addition of Methods for Event Logs.
					- Addition of methods RPC_SetLog() and RPC_SetDebug().
					- Addition of cfg.bLog flag for enable/disable of logging.
					- Fixed bug with backlash in Circular-Optimised.
	3.0.0.1			- Addition of Debug Logs in INIT sequence.
	3.0.1.0			- Introduction of new command E_MOTOR_MOVE_TYPE.TRACKING.
					- Logs are disabled while tracking.
					- GVL.C_CYCLE_IDLE set to 10 allowing a minimum of 5 NC-Task SAF cycles for each command.
					  It is assumed that PlcTask cycle time 1 ms and NC-Task SAF cycle time is 2 ms.
					- Idle command cycles are compared with FB_MA::RefCfg.nMinSkipCycles rather than GVL.C_CYCLE_IDLE.
					- Addition of FB_MA::CmdMotorMoveTrk() that sends E_MOTOR_MOVE_TYPE.TRACKING command in tracking.
					- FB_MA::User_HandleExternalCmds is the only place where RefStat.nSkippedCycles is incremented.
					- ENG and OFF buttons on FB_MA_ADC GUI send TRK_CMD_STOP_TRACK instead of TRK_CMD_MOVE.
	3.0.1.1			- Renamed TC_EVENTS.OpsEventClass to TC_EVENTS.MotorOpsEventClass.
					- The EventClas must have unique name.
					- Warning: Don't use ver. 3.0.1.0.
	3.0.2.0			- Compiled with TC3.1.4022.27.
					- Solved problem of 'growing' libraries by setting 
					  Property/Advanced/BuildAction to None for Motor.library and pdf files in dir config.
					- Corrected string display of seconds in F_RAD2DMS_STRING and F_RAD2HMS_STRING.
*)
	sDate:			STRING(16)	:= '2019-04-26';
	sDescription:	STRING(64) 	:= 'State Machine based Motor control';
	sName:			STRING(16)	:= 'FB_MOTOR';
	sPlatform:		STRING(16)	:= 'CoDeSys';
	sSynopsis:		STRING(64)	:= 'General purpose motor controller';
	nVersionMajor:	DINT		:= 4;
	nVersionMinor:	DINT		:= 1;

END_STRUCT
END_TYPE

// DUTs/Structures/Motor/T_MOTOR_INIT_STEP
TYPE T_MOTOR_INIT_STEP :
STRUCT
	nAction:	DINT; 	(* e.g. FIND_LHW *)
	lrValue1:	LREAL;	(* Normally velocity *)
	lrValue2:	LREAL;	(* Normally position *)
END_STRUCT
END_TYPE

// DUTs/Structures/Motor/T_MOTOR_MC_PARAMETER
TYPE T_MOTOR_MC_PARAMETER :
STRUCT
	nNumber:	MC_AxisParameter;
	lrValue:	LREAL;
END_STRUCT
END_TYPE

// DUTs/Structures/Motor/T_MOTOR_MOTION
TYPE T_MOTOR_MOTION :
STRUCT
	motionType:	E_MOTOR_MODE;
	position:	T_POSITION;
	speed:		T_MOTOR_SPEED;
END_STRUCT
END_TYPE

// DUTs/Structures/Motor/T_MOTOR_SIGNAL
TYPE T_MOTOR_SIGNAL :
STRUCT
	bActive:	BOOL	:= FALSE;
	bActiveLow:	BOOL	:= FALSE;
	bUsed:		BOOL	:= FALSE;
	lrPosition:	LREAL	:= 0.0;
END_STRUCT
END_TYPE

// DUTs/Structures/Motor/T_MOTOR_SPEED
TYPE T_MOTOR_SPEED :
STRUCT
	value: 		LREAL;
	direction: 	MC_Direction;
END_STRUCT
END_TYPE

// DUTs/Structures/Motor/T_MOTOR_STAT
TYPE T_MOTOR_STAT :
STRUCT
	bLocal:			BOOL	:= FALSE;			// if TRUE, device operated from PLC GUI 
	nCounter:		UDINT	:= 0;				// Alive flag - increments on every PLC cycle
	nCmdCycleCounter:	UDINT := 0;				// Number of cycles since last command
	

	nLastCommand:	E_MOTOR_COMMAND		:= E_MOTOR_COMMAND.NONE;// Last command sent to the device 

	nErrorCode: 	E_MOTOR_ERROR 		:= E_MOTOR_ERROR.OK;	// Error code 
	nRpcErrorCode: 	E_MOTOR_RPC_ERROR 	:= E_MOTOR_RPC_ERROR.OK;// RPC Error code
	nStatus: 		E_MOTOR_STATUS		:= E_MOTOR_STATUS.OK;	// Device status 

	nState:			E_MOTOR_STATE		:= E_MOTOR_STATE.NOTOP;
	nSubstate:		E_MOTOR_SUBSTATE	:= E_MOTOR_SUBSTATE.NOTOP_NOTREADY;

	nMode:			E_MOTOR_MODE 		:= E_MOTOR_MODE.POS;	// Mode of operation, POS or VEL


	sErrorText: 	STRING 	:= 'OK'; 			// Error text 
	sRpcErrorText: 	STRING 	:= 'OK'; 			// RPC Error text 
	sStatus: 		STRING 	:= 'OK'; 			// Status in textual form, e.g. 'OFF' 
	sLibVersion:	STRING	:= 'UNKNOWN';		// Library version as string, e.g. '1.2.0.0'
	
	sState:			STRING	:= 'NOT OP';
	sSubstate:		STRING	:= 'NOT READY';
	
	sActionDesc:	STRING	:= '';
	sEventDesc:		STRING	:= '';
	
	
	lrPosError:		LREAL := 0.0;	 	// Position error 
	lrPosTarget:	LREAL := 0.0;	 	// Target position adjusted to full Enc position 
	lrPosActual: 	LREAL;				// Actual position 
	lrScaleFactor:	LREAL;				// Scale [UU]/Enc
	lrVelActual: 	LREAL;				// Actual velocity 

	nBacklashStep:	DINT;	// Backlash step (1 or 2). If Backlash=0.0, motion starts from step 2.
	nInitStep:		DINT;	// Initialisation step in progress.
	nInitAction:	DINT;	// Passed to simulator to know if searching for limits
	
	// NOTE that the original Info Data is of type UINT, i.e. 16 bit unsigned.
	nInfoData1:		INT;	// Info Data 1 from Motor I/O terminal
	nInfoData2:		INT;	// Info Data 2 from Motor I/O terminal

	bAxisReady:		BOOL := FALSE;	// Flag if axis is ready
	bBrakeActive:	BOOL := FALSE;	// Flag if brake is active
	bEnabled:		BOOL := FALSE;	// Flag if axis is enabled
	bInitialised:	BOOL := FALSE;	// Flag if axis is initialised
	bInPosition:	BOOL := FALSE;	// Flag if axis is In-Position
	bStopSwitchPos:	BOOL := FALSE;	// Flag if LSTOP signal is active
	bStopSwitchNeg:	BOOL := FALSE;	// Flag if USTOP signal is active
	bLock:			BOOL := FALSE;	// Flag if motor is locked

	// Switch signals
	signals:		ARRAY [E_MOTOR_SWITCH_INDEX.LSTOP..E_MOTOR_SWITCH_INDEX.USTOP] OF T_MOTOR_SIGNAL;

	axis:			T_MOTOR_AXIS_CFG;	// Axis Config parameters - Read from TwinCAT Axis


END_STRUCT
END_TYPE

// DUTs/Structures/Motor/T_MOTOR_SWITCHES
TYPE T_MOTOR_SWITCHES :
STRUCT
(* Variables that need mapping *)
	bLSTOP:			BOOL;
	bLHW:			BOOL;
	bREF:			BOOL;
	bINDEX:			BOOL;
	bUHW:			BOOL;
	bUSTOP:			BOOL;
END_STRUCT
END_TYPE

// DUTs/Structures/Motor/T_POSITION
TYPE T_POSITION :
STRUCT
	number: LREAL;
END_STRUCT
END_TYPE

// DUTs/Structures/MultiAxis/T_MA_CFG
TYPE T_MA_CFG :
STRUCT
	nMinSkipCycles: DINT := GPL.C_CYCLE_IDLE;
	tout:           T_MA_TOUT_CFG;
	lrTrkThreshold:	LREAL	:= 1.0;	// If maximum error is < this, bTrackingOK = TRUE
END_STRUCT
END_TYPE

// DUTs/Structures/MultiAxis/T_MA_CTRL
TYPE T_MA_CTRL :
STRUCT
	nCommand:		E_MA_COMMAND	:= E_MA_COMMAND.NONE; 
	bExecute:		BOOL;
	nMode:          INT;
END_STRUCT
END_TYPE

// DUTs/Structures/MultiAxis/T_MA_SM_STAT
TYPE T_MA_SM_STAT :
STRUCT
	sState:			STRING	:= 'NOT OP';
	sSubstate:		STRING	:= 'NOT READY';
	
	nState:			E_MA_STATE		:= E_MA_STATE.NOTOP;
	nSubstate:		E_MA_SUBSTATE	:= E_MA_SUBSTATE.NOTOP_NOTREADY;
	
	sActionDesc:	STRING	:= '';
	sEventDesc:		STRING	:= '';
END_STRUCT
END_TYPE

// DUTs/Structures/MultiAxis/T_MA_STAT
TYPE T_MA_STAT :
STRUCT
	bLocal:			    BOOL	:= FALSE;	    // if TRUE, device operated from PLC GUI 
	bInitialised:		BOOL    := FALSE;		// Flag if device is initialised
	bConfigured:		BOOL    := FALSE;		// Flag indicated that pointers to FB_MOTOR are set
	bTrackingOK:		BOOL	:= FALSE;		// if TRUE, Can switch from PRESETTING to TRACKING.
	bTrackingBAD:		BOOL	:= FALSE;		// if TRUE, Should switch from TRACKING back to PRESETTING. 

	nMode:		     	INT;
	sStatus:			STRING 	:= '';			(* Status description *)
	nStatus:            DINT    := 0;
	lrPosError:         LREAL;					// Highest difference (actualPos - targetPos)

	nErrorCode: 	    DINT    := E_MOTOR_ERROR.OK;	// Error code 
	nRpcErrorCode: 	    DINT 	:= E_MOTOR_RPC_ERROR.OK;			(* RPC Error code *)
	sRpcErrorText: 	    STRING 	:= 'OK'; 			// RPC Error text 
	
	sLibVersion:        STRING  := '';          (* Motor.library version *)

	sm:                  T_MA_SM_STAT;           // State machine status
	nCycleTime:			UDINT	:= 10000;		// Cycle time in [100ns], default 1 ms
	
	nSkippedCycles: 	DINT := 20;
END_STRUCT
END_TYPE

// DUTs/Structures/MultiAxis/T_MA_TOUT_CFG
// Configuration common to all axes in the Multi-Axis (MA) system.
// Configuration is gethered by comparing configuration of individual motors.
// These poarameters cannot be set from the WS.
TYPE T_MA_TOUT_CFG :
STRUCT
	initTime:     	DINT := 60000;     // Default INIT timeout [ms]. The longest init time in the system.
	moveTime:     	DINT := 60000;     // Default MOVE timeout [ms]. The longest init time in the system.
	stopTime:     	DINT := 10000;     // Default STOP timeout [ms]. The longest init time in the system.
END_STRUCT
END_TYPE

// DUTs/Structures/Simulation/T_SIM_MOTOR_CFG
TYPE T_SIM_MOTOR_CFG :
STRUCT
	bArrActiveLow:		ARRAY [E_MOTOR_SWITCH_INDEX.LSTOP..E_MOTOR_SWITCH_INDEX.USTOP] OF T_MOTOR_ACTIVE_LOW;
	bUseBrake:			BOOL	:= FALSE;
	bActiveLowBrake:	BOOL 	:= FALSE;
	
	// Action delays
	nDelay_SwitchFind:		UDINT := 5000;	// Delay for finding switch [ms]
	nDelay_SwitchActive:	UDINT := 3000;	// Delay for switch being active (exiting switch) [ms]
	nDelay_Brake:			UDINT :=  500;	// Delay for brake activation [ms]

	nCouplerState:			UINT := 8;		// HW state
END_STRUCT
END_TYPE

// DUTs/Structures/Simulation/T_SIM_MOTOR_STAT
TYPE T_SIM_MOTOR_STAT :
STRUCT
	bInitialised:	BOOL 	:= FALSE;
	nErrorCode: 	DINT 	:= E_MOTOR_ERROR.SIM_NOT_INITIALISED;	(* Error code *)
	sErrorText: 	STRING 	:= 'NOT INITIALISED'; 			(* Error text *)
	sStatus: 		STRING 	:= 'ERROR'; 					(* motor status in textual form, e.g. 'OK' or 'ERROR'*)
END_STRUCT
END_TYPE

// DUTs/Structures/Tracking/T_ADC_CFG
TYPE T_ADC_CFG EXTENDS T_TRK_CFG :
STRUCT
	//
	// Configuration common to both ADC's.
	//
	lrPslope:       LREAL := 0.0023;		// Pressure slope [arcsec/mbar] (
	lrPoffset:		LREAL := 743.0;			// Default Pressure offset [mbar].
	lrTslope:       LREAL := -0.0061;		// Default Temperature slope [arcsec/degC]
	lrToffset:      LREAL := 12;			// Default Temperature offset [degC]
	lrAfactor:		LREAL := 3.32;			// ADC refraction factor [1/arcsec]
	lrZDlimit:      LREAL := 0.0174533;     // 1.0 deg Zenith Distance limit [rad]

	lrMinElev:      LREAL := 27.64;			// Minimum elevation [deg]


	// Specific configuration for each ADC unit, i.e. for each motor
	unitCfg:		ARRAY [1..2] OF T_ADC_UNIT_CFG;
END_STRUCT
END_TYPE

// DUTs/Structures/Tracking/T_ADC_CMD
TYPE T_ADC_CMD :
STRUCT
	motor_ctrl: T_MOTOR_CTRL;
END_STRUCT
END_TYPE

// DUTs/Structures/Tracking/T_ADC_CTRL
TYPE T_ADC_CTRL EXTENDS T_TRK_CTRL :
STRUCT
	lrTargetPos:    ARRAY [1..2] OF LREAL;
	lrTargetVel:    LREAL;
	lrPosang: 		ARRAY [1..2] OF LREAL;
END_STRUCT
END_TYPE

// DUTs/Structures/Tracking/T_ADC_INFO
TYPE T_ADC_INFO :
STRUCT
	(* Driver Information *)
	sDate:			STRING(32)	:= '2017-07-19';
	sDescription:	STRING(80) 	:= 'ADC control';
	sName:			STRING(64)	:= 'FB_ADC';
	sPlatform:		STRING(32)	:= '';
	sSynopsis:		STRING(64)	:= '';
	nVersionMajor:	DINT		:= 0;
	nVersionMinor:	DINT		:= 1;
END_STRUCT
END_TYPE

// DUTs/Structures/Tracking/T_ADC_STAT
TYPE T_ADC_STAT EXTENDS T_TRK_STAT :
STRUCT
	lrPos:			 	LREAL   := 0.0;
	lrAdaPosAngle:      LREAL   := 0.0;
	lrDrotPos:          LREAL   := 0.0;
END_STRUCT
END_TYPE

// DUTs/Structures/Tracking/T_ADC_UNIT_CFG
TYPE T_ADC_UNIT_CFG :
STRUCT
	nSignOff:   	DINT  := 1;				// sign, e.g. ADC position sign for OFF  mode
	nSignAuto:      DINT  := 1;				// sign, e.g. ADC position sign for AUTO mode
	nSignPhi: 	    DINT  := 1;				// sign, e.g. ADC sign for phi (refraction) component

	lrRefOff:       LREAL := 0.0;			// Reference (offset) for OFF  mode
	lrRefAuto:      LREAL := 0.0;			// Reference (offset) for AUTO mode

	lrCoffset:		LREAL := 1.7387;		// Default C offset [arcsec]
	lrPosOffset:    LREAL := 90;			// Default Position offset [deg]
	lrDrotFactor:   LREAL := 2;				// Derotator factor

END_STRUCT
END_TYPE

// DUTs/Structures/Tracking/T_DROT_CFG
TYPE T_DROT_CFG EXTENDS T_TRK_CFG :
STRUCT
	nFocusSign: 	DINT  := -1;             (* Sign 2 in LCU code *)
	nDirSign:   	DINT  := 1;              (* Sign 1 in LCU code *)
	lrSkyRef:    	LREAL := 0;              (* SKY reference position  *)
    lrElevRef:   	LREAL := 0;              (* ELEV reference position *)
	lrStatRef:   	LREAL := 0;              (* STAt reference position *)
	lrUserRef:   	LREAL := 0;              (* USER reference position *)
	lrUserPar1:  	LREAL := 0;				 (* User parameter 1        *)
	lrUserPar2:  	LREAL := 0;				 (* User parameter 2        *)
	lrUserPar3:  	LREAL := 0;				 (* User parameter 3        *)
	lrUserPar4:     LREAL := 0;              (* User parameter 4        *)
END_STRUCT
END_TYPE

// DUTs/Structures/Tracking/T_DROT_CTRL
TYPE T_DROT_CTRL EXTENDS T_TRK_CTRL :
STRUCT
	lrTargetPos:    LREAL;
	lrTargetVel:    LREAL;
	lrPosang: 		LREAL;
	lrUserPar1:     LREAL := 0.0;
	lrUserPar2:     LREAL := 0.0;
	lrUserPar3:     LREAL := 0.0;
	lrUserPar4:     LREAL := 0.0;
END_STRUCT
END_TYPE

// DUTs/Structures/Tracking/T_DROT_INFO
TYPE T_DROT_INFO :
STRUCT
	(* Driver Information *)
	sDate:			STRING(32)	:= '2017-07-19';
	sDescription:	STRING(80) 	:= 'Drotator control';
	sName:			STRING(64)	:= 'FB_DROT';
	sPlatform:		STRING(32)	:= '';
	sSynopsis:		STRING(64)	:= '';
	nVersionMajor:	DINT		:= 0;
	nVersionMinor:	DINT		:= 1;
END_STRUCT
END_TYPE

// DUTs/Structures/Tracking/T_DROT_STAT
TYPE T_DROT_STAT EXTENDS T_TRK_STAT :
STRUCT
	lrAngleOnSky:       LREAL   := 0;
	lrModeAngle:        LREAL   := 0;
	lrActualVel:        LREAL;
	lrPosAng:           LREAL   := 0.0;
	lrPos:			 	LREAL   := 0.0;
	lrUserPar1:         LREAL;
	lrUserPar2:         LREAL;
	lrUserPar3:         LREAL;
	lrUserPar4:         LREAL;
END_STRUCT
END_TYPE

// DUTs/Structures/Tracking/T_TRK_CFG
TYPE T_TRK_CFG EXTENDS T_MA_CFG :
STRUCT
	site:     TrkSiteConstants;
END_STRUCT
END_TYPE

// DUTs/Structures/Tracking/T_TRK_CTRL
TYPE T_TRK_CTRL EXTENDS T_MA_CTRL :
STRUCT
	environment:     TrkEnvironment;
END_STRUCT
END_TYPE

// DUTs/Structures/Tracking/T_TRK_STAT
TYPE T_TRK_STAT EXTENDS T_MA_STAT :
STRUCT
	apparent   :        TrkApparentCoordinates;
	data       :        TrkComputation;
END_STRUCT
END_TYPE

// GVLs/GVL_TrkDefaultEnvironment
{attribute 'qualified_only'}
VAR_GLOBAL
	C_HUMIDITY:    LREAL := 50.0;
	C_LAPSERATE:   LREAL := 0.0065;
	C_PRESSURE:    LREAL := 760.0;
	C_TEMPERATURE: LREAL := 20;
END_VAR

// GVLs/GVL_TrkSiteConstants
{attribute 'qualified_only'}
VAR_GLOBAL
	C_HEIGHT    : LREAL := 2648;
	C_LONGITUDE : LREAL := 1.228800386;
	C_LATITUDE  : LREAL := -0.429833092;
END_VAR

// Version/Global_Version
{attribute 'TcGenerated'}
{attribute 'no-analysis'}
{attribute 'linkalways'}
// This function has been automatically generated from the project information.
VAR_GLOBAL CONSTANT
	{attribute 'const_non_replaced'}
	stLibVersion_ESO_LDC_Motor_Library : ST_LibVersion := (iMajor := 4, iMinor := 2, iBuild := 2, iRevision := 7, nFlags := 0, sVersion := '4.2.2.7');
END_VAR

// GCL
{attribute 'qualified_only'}
VAR_GLOBAL CONSTANT
    C_PI:				LREAL := 3.1415926535897932384626433832795028841971693993751;
    C_PI2: 				LREAL := C_PI / 2.0;
	C_2PI: 				LREAL := 2.0 * C_PI;
	C_RAD2DEG:  		LREAL := (180.0 / C_PI);
	C_DEG2RAD:  		LREAL := (C_PI / 180.0);
	// pi/(12*3600):  seconds OF TIME TO radians */
	C_S2R:				LREAL := 7.2722052166430399038487115353692196393452995355905E-5;

	C_DIAG_COE_IDX: 	WORD  := 16#FA80; 	// EL_6688 CoE address for diagnostic data
	C_UTC_OFFSET_SIDX: 	BYTE  := 11;		// EL_6688 CoE subindex for UTC offset - Leap second
	C_PTP_OFFSET_SIDX: 	BYTE  := 6;			// EL_6688 Coe subindex for PTP offset from master

	C_KELVIN:			LREAL := 273.15;	// Zero deg C expressed in [deg K]
	C_MAX_P:    		LREAL := 900.0;		// Maximum pressure [mbar]
	C_MIN_P:    		LREAL := 600.0;		// Minimum pressure [mbar]
	C_MAX_T:    		LREAL := 50.0;		// Maximum temperature [deg C]
	C_MIN_T:			LREAL := -20.0;		// Minimum temperature [deg C]
	
	C_LATITUDE_ELT:		LREAL := -0.429165991;	// ELT Latitude  [rad]
	C_LATITUDE_VLT_UT1:	LREAL := -0.429833092;	// VLT_UT1 Latitude [rad] -24 deg 37 min 39.44 sec
	C_LATITUDE_VLT_UT2:	LREAL := -0.429825122;	// VLT_UT2 Latitude [rad] -24 deg 37 min 37.80 sec
	C_LATITUDE_VLT_UT3:	LREAL := -0.429819523;	// VLT_UT3 Latitude [rad] -24 deg 37 min 36.64 sec
	C_LATITUDE_VLT_UT4:	LREAL := -0.429823005;	// VLT_UT4 Latitude [rad] -24 deg 37 min 37.36 sec
	C_LATITUDE_NTT:		LREAL := -0.5106547351;	// NTT Latitude  [rad]
	C_LATITUDE_VISTA:	LREAL := -0.4296250041;	// VISTA Latitude  [rad] -24 36 56.518226
	C_LATITUDE_VST:		LREAL := -0.429788783;	// VST Latitude  [rad] -24 deg 37 min 30.300 sec
	C_LATITUDE_VLT_CM:	LREAL := -0.429833092;	// VLT_CM Latitude  [rad]

	C_LONGITUDE_ELT:	LREAL :=  1.225074527;	// ELT Longitude [rad]
	C_LONGITUDE_VLT_UT1:LREAL :=  1.228800386;	// VLT_UT1 Longitude [rad] 70 deg 24 min 18.27 sec
	C_LONGITUDE_VLT_UT2:LREAL :=  1.228796107;	// VLT_UT2 Longitude [rad] 70 deg 24 min 17.39 sec
	C_LONGITUDE_VLT_UT3:LREAL :=  1.228790929;	// VLT_UT3 Longitude [rad] 70 deg 24 min 16.32 sec
	C_LONGITUDE_VLT_UT4:LREAL :=  1.228780856;	// VLT_UT4 Longitude [rad] 70 deg 24 min 14.25 sec
	C_LONGITUDE_NTT:	LREAL :=  1.2345499197;	// NTT Longitude [rad]
	C_LONGITUDE_VISTA:	LREAL :=  1.2286692091;	// VISTA Longitude [rad] 70 23 51.216354
	C_LONGITUDE_VST:	LREAL :=  1.228759771;	// VST Longitude [rad] 70 deg 24 min 09.896 sec
	C_LONGITUDE_VLT_CM:	LREAL :=  1.228800386;	// VLT_CM Longitude [rad]

	
	C_LEAP_SECOND:		DINT  := 37;		// Last known Leap Second
	
	C_OFFSET_UNIX:		DINT  :=  946684800;  // seconds between years 1970 and 2000 


	C_CONST1:		LREAL :=  1721013.5;      // CONSTANT used in formula
	C_CONST2:		LREAL :=  190002.5;       // CONSTANT used in formula
	C_CONST3:		LREAL :=  2400000.5;      // CONSTANT used in formula
	C_CONST4:		LREAL :=  2440587.5;      // JD FOR 1970-01-01 00:00:00.000000


//#define vltMOD(A,B) ((B)!=0.0?((A)*(B)>0.0?(A)-(B)*floor_((A)/(B)):(A)+(B)*floor_(-(A)/(B))):(A))


END_VAR

// GPL
{attribute 'qualified_only'}
VAR_GLOBAL CONSTANT
	C_CYCLE_IDLE: 		DINT  := 10;		// Minimum number of idle cycles between commands to motor

    C_POS_SPEED: 		LREAL := 3;			// TODO ?
    C_MAX_SPEED: 		LREAL := 5;			// TODO ?
	C_MIN_SPEED: 		LREAL := 0.01;		// TODO ?

	C_MA_MAX_AXES:		INT 	:= 6;			// Maximum number of axes
	
END_VAR

// DUTs/Interfaces/ITrackCtrl
INTERFACE ITrackCtrl

METHOD ComputeNextPos : BOOL
VAR_INPUT
END_VAR

VAR_OUTPUT
	newPos : LREAL;
END_VAR
END_METHOD

METHOD HandleStates : BOOL
VAR_INPUT
END_VAR
END_METHOD

METHOD Init : BOOL
VAR_INPUT
END_VAR
END_METHOD

METHOD IsError : BOOL
VAR_INPUT
END_VAR
END_METHOD

METHOD MoveInPos : BOOL
VAR_INPUT
	refMotion: REFERENCE TO T_MOTOR_MOTION;
END_VAR
END_METHOD

METHOD MoveInSpeed
VAR_INPUT
	refMotion: REFERENCE TO T_MOTOR_MOTION;
END_VAR
END_METHOD

METHOD Reset : BOOL
VAR_INPUT
END_VAR
END_METHOD

END_INTERFACE

// POUs/Astro/FB_ASTRO
FUNCTION_BLOCK FB_ASTRO
VAR_INPUT
	in_equinox: 	LREAL := 2000.0;
	in_latitude:	LREAL := GCL.C_LATITUDE_ELT;
	in_longitude:	LREAL := GCL.C_LONGITUDE_ELT;
END_VAR
VAR_OUTPUT
END_VAR
VAR
	//	Physical Inputs to be mapped
	i_EL6688_Data		AT%I*: 	T_ASTRO_EL6688_DATA;	// Link to corresponding inputs of EL6688
	i_DcToTcTimeOffset	AT%I*:	LINT;					// Link to EtherCAT/InfoData/DcToTcTimeOffset
	i_DcToExtTimeOffset	AT %I*:	LINT;					// Link to EtherCAT/InfoData/DcToExtTimeOffset
	i_EL6688_AdsAddr	AT %I*:	AMSADDR;				// Leap Second ADS address structure

	//	Physical Outputs to be mapped
	q_Astro_Data		AT%Q*: 	T_ASTRO_OUTPUT;		// Link to C++ input structure 
	
	// TEL data updated from WS via OPC UA
	{attribute 'OPC.UA.DA' := '1'}
	stTel_IF:			T_ASTRO_TEL_IF;	// ra, dec, ada, corrector, etc
	
	{attribute 'OPC.UA.DA' := '1'}
//	stCoordinates:		T_ASTRO_TEL_DATA;
	
	{attribute 'OPC.UA.DA' := '1'}
	stat:				T_ASTRO_STAT;
	
	

	// Read Leap Second every time this string is found in the UTC date,
	// i.e. Read Leap Second every night one second after midnight.
	sDateCheck:			STRING := '00:00:00.999';	// '2018-09-04-07:06:17.712705664'
END_VAR

M_Configure();		// Trigger a Leap Second read

M_GetLeapSecond();	// Executed during startup and if UTC has string '00:00:00.999'

M_Update();			// Assign all outputs

METHOD M_Configure : BOOL
VAR_INPUT
END_VAR
VAR_INST
	{attribute 'OPC.UA.DA' := '0'}
	i:	INT := 0;
END_VAR
IF NOT stat.bConfigured THEN
	i	:= i + 1;
	// Delay reading of EL6688 parameters by 5 sec (1 ms cycle time)
	IF i = 5000 THEN
		// Take input parameters
		q_Astro_Data.stCoordinates.equinox	:= in_equinox;
		q_Astro_Data.stCoordinates.latitude	:= in_latitude;
		q_Astro_Data.stCoordinates.longitude:= in_longitude;
		
		// Set parameters for reading the Leap Second
		stat.sAmsNetId		:= F_CreateAmsNetId(i_EL6688_AdsAddr.netId);
		stat.nAmsPort		:= i_EL6688_AdsAddr.port;
		stat.bGetLeapSecond	:= TRUE;	// Trigger read

	END_IF

	IF stat.bLeapSecondRead THEN
		stat.bConfigured	:= TRUE;
	END_IF
ELSE
	// Read Leap Second every night just after midnight.
	// We are looking for string '00:00:00.999' at position 12 in UTC time string, 
	// e.g. in '2018-09-04-00:00:00.999705664'
	// WARNING: This only works if the cycle time is 1 ms !!!
	IF find (stat.sUtcTime, sDateCheck) = 12 THEN
		stat.bGetLeapSecond	:= TRUE;	// Trigger read
	END_IF
END_IF
END_METHOD

METHOD M_CycleUpdate : BOOL
VAR_INPUT
END_VAR
;
(*
HRESULT CTrkMod::CycleUpdate(ITcTask* ipTask, ITcUnknown* ipCaller, ULONG_PTR context)
{
	HRESULT hr = S_OK;
	AstroCoordinates coord;
	vltTIMEVAL utc;
	vltTRACK_INFO track;
	PTPTime ptpTime;

	//memcpy(&coord, &m_Inputs.stCoordinates, sizeof(AstroCoordinates));

	coord.ra = m_Inputs.stCoordinates.ra;
	coord.dec = m_Inputs.stCoordinates.dec;
	coord.equinox = m_Inputs.stCoordinates.equinox;
	coord.latitude = m_Inputs.stCoordinates.latitude;
	coord.longitude = m_Inputs.stCoordinates.longitude;

	memcpy(&ptpTime, &m_Inputs.stPtpTime, sizeof(PTPTime));

	 // Distributed clock timestamp at "begin of task" (independent from read time within task cycle)
	hr = FAILED(hr) ? hr : m_spRTime->GetCurDcTime(GETCURDCTIME_ACTUAL, &m_Outputs.stTime.dcTime );

	if (timeGetAbsoluteDcTime(ptpTime, m_Inputs.leap_second, &m_Outputs.stTime.dcTime) == S_FALSE)
			m_Outputs.stTime.mode = TIME_LOCAL;
	else
			m_Outputs.stTime.mode = TIME_UTC;
			
	timeGetUTC(m_Outputs.stTime.dcTime, &utc);
	TrkUpdate(coord, utc, track);
	m_Outputs.stTracking.alt     = track.alt;
	m_Outputs.stTracking.alt_deg = track.alt_deg;
	m_Outputs.stTracking.pa      = track.pa;
	m_Outputs.stTracking.pa_deg  = track.pa_deg;
	m_Outputs.stTracking.ha      = track.ha;
	m_Outputs.stTracking.gmst    = track.gmst;
	m_Outputs.stTracking.az      = track.az;
	m_Outputs.stTracking.az_deg  = track.az_deg;
	m_Outputs.stTracking.ra_r    = track.ra_r;
	m_Outputs.stTracking.dec_r   = track.dec_r;
	m_counter+=m_Inputs.Value;
	m_Outputs.Value=m_counter;

	return hr;
}
*)
END_METHOD

//	This method calculates the absolute time based on 
//	- the actual DC system time 
//	- Internal and External timestamps from the module EL6688
//	- DC2TC and DC2Ext offsets from EtherCAT device.
METHOD M_DcAbsoluteTime : BOOL
VAR_INPUT
END_VAR
VAR
(*	dcSysTime:		LINT;*)
	utcTime:		ULINT;
	tDc2UtcDiff:	LINT;
	tDcCurrentTime:	ULINT;
	
	one_sec:	LINT	:= 1000000000;	// 1 sec in nanosec
	
END_VAR
VAR_INST
	// Variable for testing the i_DcToExtTimeOffset term
	c:		INT := 0; 
END_VAR
(* Get current DC System Time *)
tDcCurrentTime	:= F_GetCurDcTaskTime64();

// Get DC time as STRING 
stat.sDcTime := DCTIME64_TO_STRING(tDcCurrentTime);	

(*	
	Get the UTC time

	The signal coming from the time server is TAI time, 
	i.e. includes the leap seconds.
	Our instruments work with UTC time.
	Adjust for:
		- the offset between DC and TC time.
		- the UTC leap time, i.e. add 35 secs (remove it) 
		- the time difference between external and internal time
	Note: 
	External and internal times ARE NOT current times.
	These are the values when the last reading was taken.
	It can be a couple of cycles or even seconds in the past.
	Only the difference is relevant, not the absolute values! 
*)

IF i_EL6688_Data.External_device_not_connected THEN
	// Check if external time signal is connected
	stat.bBadTimeSignal := TRUE;
ELSIF i_EL6688_Data.Internal_time_stamp = 0  OR  i_EL6688_Data.External_time_stamp = 0 THEN
	// If any timestamp is zero, it means that most probably they are not mapped.
	stat.bBadTimeSignal := TRUE;
ELSIF NOT q_Astro_Data.stUtcTime.bLeapSecondQuality THEN
	// Check if Leap Second is read correctly
	stat.bBadTimeSignal := TRUE;
ELSE
	// Checks are fine. The time signal is not bad.
	stat.bBadTimeSignal := FALSE;
END_IF


IF NOT stat.bBadTimeSignal THEN
	//
	// UTC Mode - Find the difference between DC and UTC
	//
	tDc2UtcDiff :=	ULINT_TO_LINT(i_EL6688_Data.Internal_time_stamp) - 
					ULINT_TO_LINT(i_EL6688_Data.External_time_stamp) + 
					(one_sec * q_Astro_Data.stUtcTime.nLeapSecond) +
					i_DcToTcTimeOffset + 
					c * i_DcToExtTimeOffset;
	
	stat.mode	:= E_TIME_MODE.UTC;
ELSE
	//
	// LOCAL Mode - Set the difference between DC and UTC to zero
	//
	tDc2UtcDiff := 0;

	stat.mode	:= E_TIME_MODE.LOCAL;
END_IF

// Get UTC time
utcTime	:= tDcCurrentTime - LINT_TO_ULINT(tDc2UtcDiff);
	
// Update status			
stat.tUtcTime	:= F_DCTIME64_TO_ULINT(utcTime);
stat.sUtcTime	:= DCTIME64_TO_STRING(utcTime);		// UTC time as STRING


// Assign outputs
q_Astro_Data.stUtcTime.mode				:= stat.mode;
q_Astro_Data.stUtcTime.dcTime			:= utcTime;
q_Astro_Data.stUtcTime.bBadTimeSignal	:= stat.bBadTimeSignal;
END_METHOD

METHOD M_GetLeapSecond : BOOL
VAR_INPUT
END_VAR
VAR_INST
	{attribute 'OPC.UA.DA' := '0'}
	fbSdoRead:    FB_EcCoESdoRead; (*FB FOR reading CoE objects*)
	{attribute 'OPC.UA.DA' := '0'}
	bRead:	BOOL := FALSE;
END_VAR
IF stat.bGetLeapSecond THEN
	stat.bGetLeapSecond	:= FALSE;
	
	IF stat.sAmsNetId = '0.0.0.0.0.0' OR stat.nAmsPort = 0 THEN
		q_Astro_Data.stUtcTime.bLeapSecondQuality	:= FALSE;
		q_Astro_Data.stUtcTime.nLeapSecond		:= 0;
		bRead					:= FALSE;
		stat.bLeapSecondRead	:= TRUE;
		M_GetLeapSecond			:= TRUE;
		RETURN;
	ELSE
		bRead	:= TRUE;
		// Trigger SDO read
		fbSdoRead(	sNetId		:= stat.sAmsNetId,
					nSlaveAddr 	:= stat.nAmsPort,
					nIndex 		:= GCL.C_DIAG_COE_IDX, 
					nSubIndex	:= GCL.C_UTC_OFFSET_SIDX, 
					pDstBuf 	:= ADR(stat.nLeapSecond), 
					cbBufLen 	:= SIZEOF(q_Astro_Data.stUtcTime.nLeapSecond),
					bExecute 	:= FALSE);
	END_IF
END_IF

// Read SDO for leap second
IF bRead THEN
	fbSdoRead(bExecute 	:= TRUE);
				
    IF fbSdoRead.bError THEN
		// The read has failed.
		// Probably an older version of EL6688 without GCL.C_DIAG_COE_IDX index.
		// Assume Leap Second of 0.
		bRead := FALSE;

		q_Astro_Data.stUtcTime.nLeapSecond		:= 0;
		q_Astro_Data.stUtcTime.mode				:= E_TIME_MODE.UTC;
		q_Astro_Data.stUtcTime.bLeapSecondQuality	:= TRUE;
		
		stat.bLeapSecondRead:= TRUE;
		stat.bInitialised	:= TRUE;
		M_GetLeapSecond		:= TRUE;
		;	// TODO: Handle error
	ELSIF NOT fbSdoRead.bBusy THEN
		// Reading is complete
		bRead := FALSE;

		q_Astro_Data.stUtcTime.mode			:= E_TIME_MODE.UTC;
		q_Astro_Data.stUtcTime.nLeapSecond	:= stat.nLeapSecond;
		q_Astro_Data.stUtcTime.bLeapSecondQuality	:= TRUE;
		stat.bLeapSecondRead:= TRUE;
		stat.bInitialised	:= TRUE;
		M_GetLeapSecond		:= TRUE;
	ELSE
		M_GetLeapSecond		:= FALSE;
	END_IF
END_IF
END_METHOD

METHOD M_TrkUpdate : BOOL
VAR_INPUT
END_VAR
VAR
	ra_r, dec_r:	LREAL;
	temp1, temp2, temp3, temp4:	LREAL;
	ut1, t, tu, A:	LREAL;
	
	sh, ch, cd, chcd, sp, sdcp, cp, sd, x, y, rsq:	LREAL;

	track:	REFERENCE TO T_ASTRO_TRACKING_DATA;
	coord:	REFERENCE TO T_ASTRO_TEL_DATA;
END_VAR
// Use F_vltSign()
// Use F_vltMod()
;
(*
HRESULT TrkUpdate(
						AstroCoordinates& coord, 	// FB_ASTRO::stCoordinates:		T_ASTRO_COORDS; (via OPC UA)
						vltTIMEVAL& utc,			// FB_ASTRO::q_Astro_Data.stUtcTime:	T_ASTRO_UTC_TIME;
						vltTRACK_INFO& track		// FB_ASTRO::q_Astro_Data.stTrackingData:	T_ASTRO_TRACKING_DATA;
						)
{
	HRESULT hr = S_OK;
	AstroCoordinates wc_rad;
	double temp1, temp2, temp3, temp4;
	double ut1;
	double t;
	double tu;
	double A;
	
	 wc_rad.ra = astroHms2rad(coord.ra);
	 wc_rad.dec = astroDms2rad(coord.dec);
	
	 track.ra_r  = wc_rad.ra;
	 track.dec_r = wc_rad.dec;
	 temp1 = cos_(wc_rad.dec) * tan_(coord.latitude);
	 temp2 = sin_(wc_rad.dec);
	 temp3 = temp2 * sin_(coord.latitude);
	 temp4 = cos_(wc_rad.dec) * cos_(coord.latitude);

	 ut1 = timeUTCToMJD(&utc);
	 tu = (ut1 - 51544.5) / 36525.0;
     track.gmst = vltMOD(ut1, 1.0) * vlt2PI +
                         (24110.54841 +
                          (8640184.812866 +
                           (0.093104 - 6.2e-6 * tu) * tu) * tu) * vltS2R;
     track.gmst = vltMOD(track.gmst, vlt2PI);
     if (track.gmst < 0.0)
		 track.gmst = track.gmst + vlt2PI;
     track.ha = track.gmst - (coord.longitude + coord.equinox + wc_rad.ra);

		
    /* calc. parallactic angle */
    /* t = tan(latitude) * cos(dec) - sin(dec) * cos(hourAngle); */
    t = temp1 - temp2 * cos_(track.ha);
    if (t == 0.0)
		return S_FALSE;  /* error */

    track.pa = atan_(sin_(track.ha) / t) + vltPI;
    track.pa = vltMod(vltPI2 * vltSign(t) + track.pa +
						vltPI2 , vlt2PI) +
						vltPI2 * (-vltSign(track.ha) + 1) * 
					  (vltSign(coord.dec - coord.latitude) - 1);	// TODO: ERROR coord.dec should be wc_rad.dec [rad] !!!
    if (track.pa > vltPI)
		 track.pa -= vlt2PI;

	track.pa_deg = track.pa * vltRAD2DEG;


    /* calc. telescope altitude */
    /* altitude = asin(sin(dec) * sin(latitude) + 
                       cos(dec) * cos(latitude) * cos(hourAngle)); */
    track.alt = asin_(temp3 + temp4 * cos_(track.ha));
	track.alt_deg = track.alt * vltRAD2DEG;

	/* MKI - calc. telescope azimuth */
	/* 
	* A = acos((sin(dec) - sin(altitude) * sin(latitude))
	*             ---------------------------------------
	*			      cos(altitude)*cos(latitude))
	*/
	
	double sh, ch, cd, chcd, sp, sdcp, cp, sd, x, y, rsq;

	sh = sin_(track.ha);
	ch = cos_(track.ha);
	sd = sin_(wc_rad.dec);
	cd = cos_(wc_rad.dec);
	sp = sin_(coord.latitude);
	cp = cos_(coord.latitude);
	chcd = ch * cd;
	sdcp = sd * cp;
	x = - chcd * sp + sdcp;
	y = - sh * cd;
	rsq = x *x + y * y;
	A = rsq != 0.0 ? atan2_(y,x) : 0.0;
	// The above formula assumes 0deg North and 90deg East. This
	// must be corrected for VLT conventions 0deg is South. The 
	// complete range of azimuth will be between 0-360.
	// if (A < 0.0) A += vlt2PI;
	A = - (A + vltPI);
	if (A < 0.0)
		A += vlt2PI;
	A = vltMOD(A,vlt2PI);

	track.az = A;
	track.az_deg = track.az * vltRAD2DEG;

    /* calc. fieldRotation */
    track.fr = track.pa -  track.alt;

	return hr;

}
*)

// Set references to output data structures
track REF=q_Astro_Data.stTrackingData;
coord REF=q_Astro_Data.stCoordinates;

// DPO added
// Copy ra and dec to output data structures
track.ra_hms  := coord.ra_hms;
track.dec_dms := coord.dec_dms;

// Get ra and dec in radians
track.ra_r		:= F_astroHms2rad(stTel_IF.ra_hms);
track.dec_r		:= F_astroDms2rad(stTel_IF.dec_dms);

// TODO: We assume that ra/dec are scanned from TEL in HMS/DMS format, see T_ASTRO_TEL_IF and M_Update()
ra_r	:= track.ra_r;
dec_r	:= track.dec_r;
	
temp1 := COS(dec_r) * TAN(coord.latitude);
temp2 := SIN(dec_r);
temp3 := temp2 * SIN(coord.latitude);
temp4 := COS(dec_r) * COS(coord.latitude);

// TODO: DOUBLE timeUTCToMJD(vltTIMEVAL *ut)
ut1 := F_timeUTCToMJD(F_timeGetUTC(q_Astro_Data.stUtcTime.dcTime));	// TODO: Not correct. Should be T_TIMEVAL
tu := (ut1 - 51544.5) / 36525.0;
track.gmst :=	F_vltMOD(ut1, 1.0) * GCL.C_2PI +
				(24110.54841 + (8640184.812866 + (0.093104 - 6.2E-6 * tu) * tu) * tu) * GCL.C_S2R;
track.gmst := F_vltMOD(track.gmst, GCL.C_2PI);
IF track.gmst < 0.0 THEN
	track.gmst := track.gmst + GCL.C_2PI;
END_IF
//track.ha := track.gmst - (coord.longitude + coord.equinox + ra_r);	// TODO: Check the formula
track.ha := track.gmst - (coord.longitude + ra_r);	// TODO: Check the formula

// DPO added
track.ha_deg	:= track.ha * GCL.C_RAD2DEG;
track.ha_hms	:= F_astroRad2Hms(track.ha);

// CALC. parallactic angle 
// t = tan(latitude) * cos(dec) - sin(dec) * cos(hourAngle); 
t := temp1 - temp2 * COS(track.ha);
IF t = 0.0 THEN
	M_TrkUpdate := FALSE;  // error 
	RETURN;
END_IF

// slaPa() does this differently
// Result is in the range +- PI
// TODO: Use this formula.
track.pa := F_slaPa(track.ha, dec_r, coord.latitude);

// Original PA calculation
track.pa := ATAN(SIN(track.ha) / t) + GCL.C_PI;
track.pa := F_vltMod(GCL.C_PI2 * F_vltSign(t) + track.pa + GCL.C_PI2 , GCL.C_2PI) +
					GCL.C_PI2 * (-F_vltSign(track.ha) + 1) * 
				  (F_vltSign(dec_r - coord.latitude) - 1);	// TODO: ERROR? was coord.dec_dms, should be wc_rad.dec [rad] !!!
IF track.pa > GCL.C_PI THEN
	track.pa := track.pa - GCL.C_2PI;
END_IF

track.pa_deg := track.pa * GCL.C_RAD2DEG;


// CALC. telescope altitude 
// altitude = asin(sin(dec) * sin(latitude) + cos(dec) * cos(latitude) * cos(hourAngle));
track.alt := ASIN(temp3 + temp4 * COS(track.ha));
track.alt_deg := track.alt * GCL.C_RAD2DEG;

// DPO: slaE2h()
(*
	/* MKI - CALC. telescope azimuth */
	/* 
	* A = acos((sin(dec) - sin(altitude) * sin(latitude))
	*             ---------------------------------------
	*			      cos(altitude)*cos(latitude))
	*/
*)
sh := SIN(track.ha);
ch := COS(track.ha);
sd := SIN(dec_r);
cd := COS(dec_r);
sp := SIN(coord.latitude);
cp := COS(coord.latitude);
chcd := ch * cd;
sdcp := sd * cp;
x := - chcd * sp + sdcp;
y := - sh * cd;
rsq := x *x + y * y;

// TODO: A = rsq != 0.0 ? atan2_(y,x) : 0.0;
IF rsq <> 0.0 THEN
	A := F_atan2(y,x);
ELSE
	A := 0.0;
END_IF
// The above formula assumes 0deg North and 90deg East. This
// must be corrected for VLT conventions 0deg is South. The 
// complete range of azimuth will be between 0-360.
// if (A < 0.0) A += vlt2PI;
A := - (A + GCL.C_PI);
IF A < 0.0 THEN
	A := A + GCL.C_2PI;
END_IF
A := F_vltMOD(A,GCL.C_2PI);

track.az 		:= A;
track.az_deg	:= track.az * GCL.C_RAD2DEG;

// calc. fieldRotation 
track.fr := track.pa -  track.alt;

M_TrkUpdate := TRUE;  // OK
END_METHOD

// Update the output structure q_CPP_Data that should be linked
// to the C++ module that calculates tracking data.
METHOD M_Update : BOOL
VAR_INPUT
END_VAR
// Get UTC time and Local time
M_DcAbsoluteTime();

// Update TEL location and equinox
q_Astro_Data.stCoordinates.equinox		:= stTel_IF.equinox;
q_Astro_Data.stCoordinates.latitude		:= stTel_IF.latitude;
q_Astro_Data.stCoordinates.longitude	:= stTel_IF.longitude;

// Update TEL coordinates
q_Astro_Data.stCoordinates.ra_hms		:= stTel_IF.ra_hms;
q_Astro_Data.stCoordinates.dec_dms		:= stTel_IF.dec_dms;
q_Astro_Data.stCoordinates.adaPos_deg	:= stTel_IF.adaPos_deg;
q_Astro_Data.stCoordinates.corrPos_deg	:= stTel_IF.corrPos_deg;

// Update atmospheric conditions
q_Astro_Data.stAtmosphere.lrHumidity	:= stTel_IF.lrHumidity;
q_Astro_Data.stAtmosphere.lrPressure	:= stTel_IF.lrPressure;
q_Astro_Data.stAtmosphere.lrTemperature	:= stTel_IF.lrTemperature;

// Update tracking data, i.e. gmst, ra, dec, alt, az, pa, ha, etc.
M_TrkUpdate();
END_METHOD

END_FUNCTION_BLOCK

// POUs/Functions/F_DCTIME64_TO_ULINT
FUNCTION F_DCTIME64_TO_ULINT : ULINT
VAR_INPUT
	in:		T_DCTIME64;
END_VAR
VAR
	out:	ULINT;
END_VAR

memcpy (ADR(out), ADR(in), SIZEOF(in));
F_DCTIME64_TO_ULINT	:= out;

END_FUNCTION

// POUs/Functions/F_vltSign
FUNCTION F_vltSign : LREAL
VAR_INPUT
	number:	LREAL;
END_VAR
VAR
END_VAR

(*
static double vltSign(double number)
{
    if (number >= 0)
	return 1.0;
    return -1.0;
}
*)

IF number >= 0 THEN
	F_vltSign	:= 1.0;
ELSE
	F_vltSign	:= -1.0;
END_IF

END_FUNCTION

// POUs/Functions/F_vltMod
FUNCTION F_vltMod : LREAL
VAR_INPUT
	number:		LREAL;
	divisor:	LREAL;
END_VAR
VAR
END_VAR

(*
static double vltMod(double number, double divisor)
{
    if (divisor == 0.0)
	return 0.0;
    return number - divisor * (int) (number / divisor);
}


*)

IF divisor = 0.0 THEN
	F_vltMod	:= 0.0;
ELSE
	F_vltMod	:= number - divisor * TRUNC_INT(number / divisor);
END_IF

END_FUNCTION

// POUs/Functions/F_astroHms2rad
(*
 *   astroHms2rad   :   Convert a time/angle,given in user format, to radians.
 *   ===========
 *
 *   Given    :  angle      an angle as hhmmss.ttt (HoursMinutesSecs)
 *   Returned :  rad        the angle as radians
 *
 *    The given time/angle, a floating value in the format HHMMSS.TTT, is 
 *    converted to radians. See also tcsSplitHms
 *)
FUNCTION F_astroHms2rad : LREAL
VAR_INPUT
	angle:	LREAL;
END_VAR
VAR
	hh,hm,hs:	LREAL;
	rad,rar:	LREAL;
END_VAR

(*
double astroHms2rad (double angle)
{
   double hh,hm,hs;
   double rad,rar;
   double de2ra = 0.017453292519943;

   astroSplitHms(fabs_(angle),&hh,&hm,&hs);
   rad=(hh + hm/60.0 + hs/3600.0)*15.0;
   rar=rad*de2ra;
   if (angle<0.0) rar=-rar;
   
   return(rar);
}

*)

F_astroSplitHms(ABS(angle),h=>hh,m=>hm,sec=>hs);

rad	:= (hh + hm/60.0 + hs/3600.0) * 15.0;	// * 15.0 : 24h * 15 = 360 deg
rar	:= rad * GCL.C_DEG2RAD;

IF angle<0.0 THEN
	rar := -rar;
END_IF

F_astroHms2rad	:= rar;

END_FUNCTION

// POUs/Functions/F_astroSplitHms
(*
 *   tcsSplitHms   :   Split an angle,given in user format, to its
 *   ===========      parts.
 *
 *   Given    :  angle      an angle as hhmmss.ttt (or ddmmss.tt)
 *   Returned :  h          hours (degrees)
 *               m          minutes (arcminutes)
 *               s          seconds (arcseconds)
 *
 *    The given time/angle, a floating value in the format HHMMSS.TTT, is split
 *    up in the parts HH, MM and SS.TTT (or DDMMSS.TTT if the input parameter
 *    is an angle).  
 *          NOTE:   if the given value is negative, all returned values 
 *    will also be negative! Which is may be not what you want, so take care of
 *    the sign outside of this function!
 * 
 *
 *   EXAMPLES
 *    Example 1:
 *     double time,h,m,s;
 *     time=123456.7;
 *     i=astroSplitHms(time,&h,&m,&s);
 *
 *        will return  h=12.0
 *                     m=34.0
 *                     s=56.7 
 *
 *
 *   Example 2:
 *     double time,h,m,s;
 *     time=345.0;
 *     i=astroSpltHms(time,&h,&m,&s);
 *
 *        will return  h=0.0
 *                     m=3.0
 *                     s=45.0 
 *
 *)
FUNCTION F_astroSplitHms : bool
VAR_INPUT
	angle:	LREAL;	// an angle as hhmmss.ttt (or ddmmss.tt)
END_VAR
VAR_OUTPUT
	h, m, sec:	LREAL;
END_VAR
VAR
   val:	LREAL;
   hours,minutes,seconds,t1,t2,t3:	LREAL;
 END_VAR

(*
void astroSplitHms (double angle, double *h, double *m, double *s)
{
   double val;
   double hour,min,sec,t1,t2,t3;
   
   val  = angle;  
   sec  = val - (int)(val/100.0)*100.0;    
   t1   = val-sec;
   t2   = t1 - (int)(t1/10000.0)*10000.0;
   min  = t2/100.0;
   t3   = val-sec-t2;
   hour = t3/10000;
   *h   = hour;
   *m   = min;
   *s   = sec;   
   return;
}
*)

val		:= angle;  
seconds	:= val - TRUNC_INT(val/100.0) * 100.0;    
t1		:= val - seconds;
t2		:= t1 - TRUNC_INT(t1/10000.0) * 10000.0;
minutes	:= t2/100.0;
t3		:= val - seconds - t2;
hours	:= t3/10000;

h	:= hours;
m	:= minutes;
sec	:= seconds;   

F_astroSplitHms	:= TRUE;

END_FUNCTION

// POUs/Functions/F_astroDms2rad
(*
 *   astroDms2rad   :   Convert an angle,given in user format, to radians.
 *   ===========
 *
 *   Given    :  angle      an angle as ddmmss.ttt (DegreesMinutesSecs)
 *   Returned :  rad        the angle as radians
 *
 *    The given angle, a floating value in the format DDMMSS.TTT, is 
 *    converted to radians. See also tcsSplitHms.
 *)
FUNCTION F_astroDms2rad : LREAL
VAR_INPUT
	angle:	LREAL;
END_VAR
VAR
	hh,hm,hs:	LREAL;
	ded,der:	LREAL;
END_VAR

(*
double astroDms2rad (double angle)
{
   double hh,hm,hs;
   double ded,der;
   double de2ra = 0.017453292519943;

   astroSplitHms(fabs_(angle),&hh,&hm,&hs);
   ded=hh + hm/60.0 + hs/3600.0;
   if (angle<0.0) ded=-ded; 
   der=ded*de2ra;
   
   return(der);
}*)

F_astroSplitHms(ABS(angle),h=>hh,m=>hm,sec=>hs);

ded	:= hh + hm/60.0 + hs/3600.0;

IF angle<0.0 THEN
	ded := -ded;
END_IF

der	:= ded * GCL.C_DEG2RAD;


F_astroDms2rad	:= der;

END_FUNCTION

// POUs/Functions/F_timeUTCToMJD
(*
/*
 *****************************************************************************
 * timeUTCToMJD: convert struct ccsTIMEVAL into modified Julian date
 *
 *  IN   ut: time in UT
 *  OUT    : Modified julian date 
 ***************************************************************************** 
 */
*)
FUNCTION F_timeUTCToMJD : LREAL
VAR_INPUT
	ut:	T_TIMEVAL;
END_VAR
VAR
	mjd:	LREAL;
END_VAR

(*
DOUBLE timeUTCToMJD(vltTIMEVAL *ut)   /* time in UT                       */
    {
    DOUBLE mjd;                       /* modified julian date             */
   /*
    *# Get Julian Date from UT 
    */
    mjd = timeUTCToJD(ut);
    
   /*
    *# Convert Julian Date into Modified Julian Date according to the formula:
    *# MJD = JD - 2400000.5;
    */
    mjd-= CONST3;
    return(mjd);    
    }
*)

// Get Julian Date from UT 
mjd := F_timeUTCToJD(ut);

(*
*# Convert Julian Date into Modified Julian Date according to the formula:
*# MJD = JD - 2400000.5;
*)
F_timeUTCToMJD	:= mjd - GCL.C_CONST3;

END_FUNCTION

// POUs/Functions/F_timeUTCToJD
(*
/*
 *****************************************************************************
 * timeUTCToJD: convert struct ccsTIMEVAL into Julian date
 *
 *  IN   ut: time in UT
 *  OUT    : Julian date  
 ***************************************************************************** 
 */
*)
FUNCTION F_timeUTCToJD : LREAL
VAR_INPUT
	ut:	T_TIMEVAL;
END_VAR
VAR
END_VAR

(*
DOUBLE timeUTCToJD(vltTIMEVAL *ut)    /* time in UT                       */
    {
    DOUBLE jd;
    
   /*
    * CONST4 = jd(70-01-01 00:00:00.000000)
    */
    jd = CONST4 + (ut->tv_sec + ut->tv_usec/1000000.)/86400.;
    return(jd);
    }
*)

F_timeUTCToJD := GCL.C_CONST4 + (UDINT_TO_REAL(ut.tv_sec) + DINT_TO_REAL(ut.tv_usec)/1000000.0)/86400.0;

END_FUNCTION

// POUs/Functions/F_timeGetUTC
(*
 *****************************************************************************
 * timeGetUTC: Get UTC time from TwinCAT DC time
 *
 *  IN   dcTime: TwinCAT DC time
 *  OUT  vltUTC: UTC time 
 ***************************************************************************** 
 *)
FUNCTION F_timeGetUTC : T_TIMEVAL
VAR_INPUT
	dcTime:   ULINT;
END_VAR
VAR
	ut:	T_TIMEVAL;
END_VAR

(*
HRESULT timeGetUTC(LONGLONG dcTime, vltTIMEVAL *vltUTC)
{
	HRESULT hr = S_OK; 
	
	// DC time is in nano seconds
	vltUTC->tv_sec = (LONGLONG)(dcTime/1000000000);
	vltUTC->tv_usec = (dcTime - (vltUTC->tv_sec * 1000000000))/1000;
	
	// Added offset between year 1970 and 2000 needed by the different references
	// used in UNIX and TWINCAT
	vltUTC->tv_sec += OFFSET_UNIX;
	return hr; 
}
*)

// DC time is in nano seconds
ut.tv_sec := ULINT_TO_UDINT(dcTime/1000000000);
ut.tv_usec := ULINT_TO_DINT((dcTime - UDINT_TO_ULINT(ut.tv_sec) * 1000000000)/1000);

// Added offset between year 1970 and 2000 needed by the different references
// used in UNIX and TWINCAT
ut.tv_sec := (ut.tv_sec + DINT_TO_UDINT(GCL.C_OFFSET_UNIX));

F_timeGetUTC	:= ut;

END_FUNCTION

// POUs/Functions/F_astroRad2Hms
FUNCTION F_astroRad2Hms : LREAL
VAR_INPUT
	hh:	LREAL;	// angle in radians
END_VAR
VAR
	value:		LREAL;
	hours:		INT;
	minutes:	INT;
	seconds:	LREAL;
	
	sign:	int := 1;
END_VAR

IF hh < 0.0 THEN
	sign	:= -1;
	hh		:= -hh;
END_IF

value := hh / GCL.C_2PI * 24.0; 	// rad to hours


hours	:= TRUNC_INT(value);
minutes := TRUNC_INT((value - hours)*60.0);
seconds := (value - hours - minutes/60.0)*3600.0;

hours	:= hours * sign;	// put back the sign

					
F_astroRad2Hms	:= hours * 10000 + minutes * 100 + seconds;

END_FUNCTION

// POUs/Functions/F_slaPa
(*
/*+
**  - - - - - -
**   s l a P a
**  - - - - - -
**
**  HA, Dec to Parallactic Angle.
**
**  (double precision)
**
**  Given:
**     ha     d     hour angle in radians (geocentric apparent)
**     dec    d     declination in radians (geocentric apparent)
**     phi    d     observatory latitude in radians (geodetic)
**
**  The result is in the range -pi to +pi
**
*)
FUNCTION F_slaPa : LREAL
VAR_INPUT
	ha, dec, phi:	LREAL;
END_VAR
VAR
	cp, cqsz, sqsz:	LREAL;
	result:			LREAL;
END_VAR

(*
{
   double cp, cqsz, sqsz;

   cp = cos ( phi );
   sqsz = cp * sin ( ha );
   cqsz = sin ( phi ) * cos ( dec) - cp * sin ( dec) * cos ( ha );
   return ( ( sqsz != 0.0 || cqsz != 0.0 ) ? atan2 ( sqsz, cqsz ) : 0.0 );
}
*)

cp := COS ( phi );
sqsz := cp * SIN ( ha );
cqsz := SIN ( phi ) * COS ( dec) - cp * SIN ( dec) * COS ( ha );

//   return ( ( sqsz != 0.0 || cqsz != 0.0 ) ? atan2 ( sqsz, cqsz ) : 0.0 );
IF sqsz <> 0.0 OR cqsz <> 0.0 THEN
	result	:= F_atan2(sqsz, cqsz);
ELSE
	result	:= 0.0;
END_IF
	
F_slaPa	:= result;

END_FUNCTION

// POUs/Functions/F_atan2
// atan2(y,x)
FUNCTION F_atan2 : LREAL
VAR_INPUT
	y:	LREAL;
	x:	LREAL;
END_VAR
VAR
	atan2val:	LREAL;
END_VAR

IF (x > 0) THEN
	atan2val := ATAN(y/x);
ELSIF ((x < 0) AND (y >= 0)) THEN
	atan2val := ATAN(y/x) + GCL.C_PI;
ELSIF ((x < 0) AND (y < 0)) THEN
	atan2val := ATAN(y/x) - GCL.C_PI;
ELSIF ((x = 0) AND (y > 0)) THEN
	atan2val := GCL.C_PI2;
ELSIF ((x = 0) AND (y < 0)) THEN
	atan2val := -GCL.C_PI2;
ELSIF ((x = 0) AND (y = 0)) THEN
	atan2val := 1000;  //represents undefined
END_IF             

F_atan2	:= atan2val;

END_FUNCTION

// POUs/CCS/FB_CCS_SIM
FUNCTION_BLOCK FB_CCS_SIM
VAR_INPUT
END_VAR
VAR_OUTPUT
END_VAR
VAR
	{attribute 'OPC.UA.DA' := '1'}
	cfg:				T_CCS_CFG;
	{attribute 'OPC.UA.DA' := '1'}
	ctrl:				T_CCS_CTRL;
	{attribute 'OPC.UA.DA' := '1'}
	stat:				T_CCS_STAT;
	
    // Tracking data structure are defined in C++ module
	{attribute 'OPC.UA.DA' := '0'}
	i_trk_data          AT %I*: TrackingData;
	
	{attribute 'OPC.UA.DA' := '0'}
	q_ccs_data          AT %Q*: CcsData;
	
	{attribute 'OPC.UA.DA' := '0'}
	q_mean_coordinates  AT %Q*: TrkMeanCoordinates;
	
END_VAR


// Get parameters
GetParams();

// Set parameters
SetParams();

METHOD FB_init : BOOL
VAR_INPUT
	bInitRetains : BOOL; // if TRUE, the retain variables are initialized (warm start / cold start)
	bInCopyCode : BOOL;  // if TRUE, the instance afterwards gets moved into the copy code (online change)
END_VAR

cfg.site.height              := GVL_TrkSiteConstants.C_HEIGHT;
cfg.site.latitude            := GVL_TrkSiteConstants.C_LATITUDE;
cfg.site.longitude           := GVL_TrkSiteConstants.C_LONGITUDE;
ctrl.environment.humidity    := GVL_TrkDefaultEnvironment.C_HUMIDITY;
ctrl.environment.lapserate   := GVL_TrkDefaultEnvironment.C_LAPSERATE;
ctrl.environment.pressure    := GVL_TrkDefaultEnvironment.C_PRESSURE;
ctrl.environment.temperature := GVL_TrkDefaultEnvironment.C_TEMPERATURE;
ctrl.meanCoordinates.alpha   := 0;
ctrl.meanCoordinates.delta   := -890000.0;
ctrl.meanCoordinates.equinox := 2000.0;
END_METHOD

METHOD GetParams
VAR_INPUT
END_VAR

// Assign output variables according input configuration and control.
memcpy(ADR(q_ccs_data.site), ADR(cfg.site), SIZEOF(q_ccs_data.site));	
memcpy(ADR(q_ccs_data.environment), ADR(ctrl.environment), SIZEOF(q_ccs_data.environment));
memcpy(ADR(q_mean_coordinates), ADR(ctrl.meanCoordinates), SIZEOF(q_mean_coordinates));
q_ccs_data.equinox := ctrl.equinox;
END_METHOD

{attribute 'TcRpcEnable':='1'}
METHOD RPC_SetCoordinates : BOOL
VAR_INPUT
	in_alpha:	 LREAL := 000000.0;
	in_delta:    LREAL := 000000.0;
	in_equinox:  LREAL := 2000.0;
END_VAR

ctrl.meanCoordinates.alpha := in_alpha;
ctrl.meanCoordinates.delta := in_delta;
ctrl.meanCoordinates.equinox := in_equinox;
END_METHOD

METHOD SetParams
VAR_INPUT
END_VAR

memcpy(ADR(stat.apparent), ADR(i_trk_data.apparent), SIZEOF(stat.apparent));
memcpy(ADR(stat.observed), ADR(i_trk_data.observed), SIZEOF(stat.observed));
memcpy(ADR(stat.data), ADR(i_trk_data.computation), SIZEOF(stat.data));

stat.lDcTime := i_trk_data.utctime.dc_time;
stat.nTimeMode := i_trk_data.utctime.mode;
IF stat.nTimeMode = 0 THEN
	stat.sTimeMode := 'Local';
ELSIF stat.nTimeMode = 1 THEN
	stat.sTimeMode := 'UTC';
ELSIF stat.nTimeMode = 2 THEN
	stat.sTimeMode := 'Simulation';
END_IF

stat.sDcTime := DCTIME64_TO_STRING(LINT_TO_ULINT(stat.lDcTime));
END_METHOD

END_FUNCTION_BLOCK

// POUs/Functions/F_MOD
FUNCTION F_MOD : LREAL
VAR_INPUT
	A:	LREAL;
	B:	LREAL;
END_VAR
VAR
END_VAR

(*
#define vltMOD(A,B) 
((B)!=0.0?
	((A)*(B)>0.0?
		(A)-(B)*floor((A)/(B))
	else
		:(A)+(B)*floor(-(A)/(B)))
else
	:(A))
*)
IF B = 0.0 THEN
	F_MOD	:= A;
ELSE
	IF A * B >= 0.0 THEN
		F_MOD	:= A - B * TRUNC_INT(A / B);
	ELSE
		F_MOD	:= A + B * TRUNC_INT(-A / B);
	END_IF
END_IF

END_FUNCTION

// POUs/Functions/F_RAD2DMS_STRING
FUNCTION F_RAD2DMS_STRING : STRING
VAR_INPUT
	dec:	LREAL;
END_VAR
VAR
	value:		LREAL;
	degrees:	INT;
	minutes:	INT;
	seconds:	LREAL;
	
	sign:	int := 1;
	result:	STRING := '';
	
	fbFormat   : FB_FormatString;
END_VAR

IF dec < 0.0 THEN
	sign	:= -1;
	dec		:= -dec;
END_IF

value := dec * GCL.C_RAD2DEG; 	// rad to hours


degrees	:= TRUNC_INT(value);
minutes := TRUNC_INT((value - degrees)*60.0);
seconds := (value - degrees - minutes/60.0)*3600.0;

// We the calculation so far the value of 14.999999999 will result
// in 14:59:60.
// We want to correct it to 15:00:00.
IF seconds > 59.999 THEN
	seconds	:= 0.0;
	minutes	:= minutes + 1;
	IF minutes = 60 THEN
		minutes	:= 0;
		degrees	:= degrees + 1;
	END_IF
// Seconds should never be < 0.0. However, it happens due to rounding
// and the value could be ~ -1.0 e-12.
// Set it to zero in that case.
ELSIF seconds < 0.0 THEN
	seconds := 0.0;
END_IF

degrees	:= degrees * sign;	// put back the sign

// format a string like "+07:01:02.123"
fbFormat( sFormat  := '%+.3d:%.2d:%06.3f', 
					arg1 := F_INT(degrees), 
					arg2 := F_INT(minutes), 
					arg3 := F_LREAL(seconds),
					sOut => result);
					
F_RAD2DMS_STRING	:= result;

END_FUNCTION

// POUs/Functions/F_RAD2HMS_STRING
FUNCTION F_RAD2HMS_STRING : STRING
VAR_INPUT
	hh:	LREAL;
END_VAR
VAR
	value:		LREAL;
	hours:		INT;
	minutes:	INT;
	seconds:	LREAL;
	
	sign:	int := 1;
	result:	STRING := '';
	
	fbFormat   : FB_FormatString;
END_VAR

IF hh < 0.0 THEN
	sign	:= -1;
	hh		:= -hh;
END_IF

value := hh / GCL.C_2PI * 24.0; 	// rad to hours


hours	:= TRUNC_INT(value);
minutes := TRUNC_INT((value - hours)*60.0);
seconds := (value - hours - minutes/60.0)*3600.0;

// We the calculation so far the value of 14.999999999 will result
// in 14:59:60.
// We want to correct it to 15:00:00.
IF seconds > 59.999 THEN
	seconds	:= 0.0;
	minutes	:= minutes + 1;
	IF minutes = 60 THEN
		minutes	:= 0;
		hours	:= hours + 1;
	END_IF
// Seconds should never be < 0.0. However, it happens due to rounding
// and the value could be ~ -1.0 e-12.
// Set it to zero in that case.
ELSIF seconds < 0.0 THEN
	seconds := 0.0;
END_IF

hours	:= hours * sign;	// put back the sign

// format a string like "+07:01:02.123"
fbFormat( sFormat  := '%+.2d:%.2d:%06.3f', 
					arg1 := F_INT(hours), 
					arg2 := F_INT(minutes), 
					arg3 := F_LREAL(seconds),
					sOut => result);
					
F_RAD2HMS_STRING	:= result;

END_FUNCTION

// POUs/Functions/F_timeGetAbsoluteDcTime
(*
 *****************************************************************************
 * timeGetAbsoluteDcTime: Adjust DC time based on the external time signal
 *
 *  IN   ptptime    : External time signal
 *  IN   leapSecond : Leap Second 
 *  OUT  dcTIME     : Adjusted TwinCAT DC time
 ***************************************************************************** 
 *)
FUNCTION F_timeGetAbsoluteDcTime : BOOL
VAR_INPUT
	ptptime:			T_ASTRO_EL6688_DATA;
	nLeapSecond:		DINT;
	DcToExtTimeOffset:	LINT;
END_VAR
VAR_IN_OUT
	dcTime:   ULINT;
END_VAR
VAR
	val:		LINT	:= 0;
	diff:		LINT	:= 0;
	one_sec:	LINT	:= 1000000000;
END_VAR

(*
HRESULT timeGetAbsoluteDcTime(PTPTime ptptime, INT leapSecond, LONGLONG *dcTime)
{
	HRESULT hr = S_OK; 
	LONGLONG val = 0;
	LONGLONG diff = 0;
	LONGLONG ONE_SEC = 1000000000;
	
	// Check if external time signal is connected
	if (ptptime.not_connected)
		return S_FALSE;

	// If both variables are null means most probably they are not mapped.
	if (ptptime.internal == 0 || ptptime.external == 0)
		return S_FALSE;

	diff = (ptptime.internal - ptptime.external) + (ONE_SEC * leapSecond) + ptptime.dcTcOffset;
	*dcTime -=  diff;
	return hr;
}*)

// Check if external time signal is connected
IF ptptime.External_device_not_connected THEN
	F_timeGetAbsoluteDcTime := FALSE;
END_IF

// If both variables are null means most probably they are not mapped.
// TODO: Is it OR or AND ?
IF ptptime.Internal_time_stamp = 0  OR  ptptime.External_time_stamp = 0 THEN
	F_timeGetAbsoluteDcTime := FALSE;
END_IF

diff := (ULINT_TO_LINT(ptptime.Internal_time_stamp) - ULINT_TO_LINT(ptptime.External_time_stamp)) + 
		(one_sec * nLeapSecond) + DcToExtTimeOffset;

dcTime	:= dcTime - LINT_TO_ULINT(diff);

F_timeGetAbsoluteDcTime := TRUE;

END_FUNCTION

// POUs/Functions/F_timeGetDcTime
(*
 *****************************************************************************
 * timeGetDcTime: Get TwinCAT DC time from UTC time
 *
 *  IN   vltUTC: UTC time 
 *  OUT  dcTIME: TwinCAT DC time
 ***************************************************************************** 
 *)
FUNCTION F_timeGetDcTime : ULINT
VAR_INPUT
	ut:	T_TIMEVAL;
END_VAR
VAR
	val:   	ULINT := 0;
END_VAR

(*
HRESULT timeGetDcTime(vltTIMEVAL vltUTC, LONGLONG *dcTime)
{
	HRESULT hr = S_OK; 
	LONGLONG val = 0;
	val = vltUTC.tv_sec * 1000000000;
	val -= OFFSET_UNIX;
	*dcTime = val + vltUTC.tv_usec * 1000;
	return hr;
}
*)
val	:= ut.tv_sec * 1000000000;
val := val - DINT_TO_ULINT(GCL.C_OFFSET_UNIX);

F_timeGetDcTime	:= val + DINT_TO_ULINT(ut.tv_usec) * 1000;

END_FUNCTION

// POUs/Motor/FB_MOTOR
FUNCTION_BLOCK FB_MOTOR EXTENDS FB_MOTOR_BASE
VAR_INPUT
	{attribute 'OPC.UA.DA' := '0'}
	sName:			STRING	:= 'Motor';	(* Default Motor name *)
	{attribute 'OPC.UA.DA' := '0'}
	nNOVRAM_DevId:	UDINT	:= 0;		(* NOVRAM device ID - normally 4 *)
	{attribute 'OPC.UA.DA' := '0'}
	nNOVRAM_Offset:	UDINT	:= 0;		(* NOVRAM offset where motor configuration is stored *)
END_VAR
VAR_OUTPUT
END_VAR
VAR
	
	(***** Local variables *****)
	{attribute 'OPC.UA.DA' := '0'}
	toutCmd:	TON;
	{attribute 'OPC.UA.DA' := '0'}
	trg:		R_TRIG;
	{attribute 'OPC.UA.DA' := '0'}
	timer:		TON;	(* Timer for measuring duration of events *)
	{attribute 'OPC.UA.DA' := '0'}
	nState_Init:			INT := MOTOR_INIT_STATE_RESET;		// State of ActivityInitializing
	{attribute 'OPC.UA.DA':='0'}
	nState_Reset:			INT := MOTOR_RESET_STATE_START;
	{attribute 'OPC.UA.DA':='0'}
	nState_PreInit:			INT	:= MOTOR_PRE_INIT_STATE_START;
	{attribute 'OPC.UA.DA':='0'}
	nState_InitSeq:			INT := MOTOR_INIT_SEQ_STATE_START;
	{attribute 'OPC.UA.DA':='0'}
	nState_PostInit:		INT	:= MOTOR_POST_INIT_STATE_START;
	{attribute 'OPC.UA.DA':='0'}
	nState_Moving:			INT := MOTOR_MOVING_STATE_WAIT_BRAKES;		// State of ActivityMoving
	{attribute 'OPC.UA.DA':='0'}
	nState_MovingNext:		INT := MOTOR_MOVING_STATE_WAIT_ABSOLUTE;	// Next state after checking brakes


	(***** Physical signals - to be mapped!!! *****)

	(* Outputs *)
	{attribute 'OPC.UA.DA' := '0'}
	q_bBrake_Ctrl	AT %Q*:	BOOL;				(* Brake control signal - DIGITAL OUT *)


	(* Inputs *)	
	{attribute 'OPC.UA.DA':='0'}
	switches		AT %I*:	T_MOTOR_SWITCHES;	(* Limit switches *)
	{attribute 'OPC.UA.DA':='0'}
	i_bInPos		AT %I*:	BOOL;				(* In-position signal - DIGITAL IN *)
	{attribute 'OPC.UA.DA':='0'}
	i_bBrake_Stat	AT %I*:	BOOL;				(* Brake feedback signal - DIGITAL IN *)
	{attribute 'OPC.UA.DA':='0'}
	i_nInfoData1	AT %I*:	UINT;				(* Info data 1 from Motor I/O terminal *)
	{attribute 'OPC.UA.DA':='0'}
	i_nInfoData2	AT %I*:	UINT;				(* Info data 2 from Motor I/O terminal *)
	{attribute 'OPC.UA.DA':='0'}
	i_nSoE_DriveStatus	AT %I*:	UINT;			(* Drive Status. SoE Drives, e.g. AX5000, ONLY!!! *)
	{attribute 'OPC.UA.DA':='0'}
	i_nSoE_PowerStatus	AT %I*:	INT;			(* Power Status. SoE Drives, e.g. AX5000, ONLY!!! *)

	{attribute 'OPC.UA.DA' := '0'}
	i_nCouplerState	AT %I*: 		UINT;	(* Link it to Coupler->InfoData->State *)

	{attribute 'OPC.UA.DA' := '0'}
	Axis:  		AXIS_REF;


(* Ctrl parameters used by ctrl.bExecute *)
	{attribute 'OPC.UA.DA':='0'}
	nCurDirection:	DINT	:=	INT_TO_DINT(MC_Positive_Direction);
	{attribute 'OPC.UA.DA':='0'}
	lrCurVelocity:	LREAL	:=	0.0;
	

(* Function block instances *)

	{attribute 'OPC.UA.DA' := '0'}
	fbHalt: 	           		MC_Halt;
	{attribute 'OPC.UA.DA' := '0'}
	fbSoEReset: 	           	FB_SoEReset;
	{attribute 'OPC.UA.DA' := '0'}
	fbResetError: 	           	MC_Reset;
	{attribute 'OPC.UA.DA' := '0'}
	fbMovePos_1:  	 			MC_MoveAbsolute;
	{attribute 'OPC.UA.DA' := '0'}
	fbMovePos_2:  	 			MC_MoveAbsolute;
	{attribute 'OPC.UA.DA' := '0'}
	ptr_fbMovePos: POINTER TO 	MC_MoveAbsolute := ADR(fbMovePos_1);
	{attribute 'OPC.UA.DA' := '0'}
	fbMoveVel_1:  	 			MC_MoveVelocity;
	{attribute 'OPC.UA.DA' := '0'}
	fbMoveVel_2:				MC_MoveVelocity;
	{attribute 'OPC.UA.DA' := '0'}
	ptr_fbMoveVel: POINTER TO 	MC_MoveVelocity := ADR(fbMoveVel_1);
	{attribute 'OPC.UA.DA' := '0'}
	fbMoveOpt_1:				MC_MoveModulo;
	{attribute 'OPC.UA.DA' := '0'}
	fbMoveOpt_2:				MC_MoveModulo;
	{attribute 'OPC.UA.DA' := '0'}
	ptr_fbMoveOpt: POINTER TO 	MC_MoveModulo := ADR(fbMoveOpt_1);
	{attribute 'OPC.UA.DA' := '0'}
	fbStop:						MC_Stop;
	{attribute 'OPC.UA.DA' := '0'}
	fbSetActualPosition:		MC_SetPosition;

	(* There are two FB's per Pos, Vel and circular-optimised. Keep track which one is active. *)
	{attribute 'OPC.UA.DA':='0'}
	nFbPos:		INT := 1; 
	{attribute 'OPC.UA.DA':='0'}
	nFbVel:		INT := 1; 
	{attribute 'OPC.UA.DA':='0'}
	nFbOpt:		INT := 1; 
	
	(* Temporary vars for finding shortest way for circular-optimised with backlash compensation *)
	{attribute 'OPC.UA.DA':='0'}
	nOptDir:		MC_Direction;	(* Optimised direction *)
	{attribute 'OPC.UA.DA':='0'}
	lrTmpDist1:		LREAL;
	{attribute 'OPC.UA.DA':='0'}
	lrTmpDist2:		LREAL;
	{attribute 'OPC.UA.DA':='0'}
	lrTmpPos1:		LREAL;
	{attribute 'OPC.UA.DA':='0'}
	lrTmpPos2:		LREAL;
	
	(* NOVRAM Handling *)
	{attribute 'OPC.UA.DA':='0'}
	bNOVRAM_Error:		BOOL := FALSE;	(* NOVRAM error active flag *)
	{attribute 'OPC.UA.DA':='0'}
	bNOVRAM_Loaded:		BOOL := FALSE;	(* Flag if NOVRAM has been loaded *)
	{attribute 'OPC.UA.DA':='0'}
	nNOVRAM_State_R:	UINT := 0;		(* NOVRAM Read state *)
	{attribute 'OPC.UA.DA':='0'}
	nNOVRAM_State_W:	UINT := 0;		(* NOVRAM Write state *)
	{attribute 'OPC.UA.DA':='0'}
	stMotorCfg_NOVRAM:	T_MOTOR_CFG;	(* NOVRAM copy of motor config. Read on First PLC cycle. *)

	{attribute 'OPC.UA.DA':='0'}
	fbNovReadWrite: 	Tc2_IoFunctions.FB_NovRamReadWriteEx;

END_VAR

// Basic configuration, executed once internally
M_Configure();

// Increment alive counter
stat.nCounter	:= stat.nCounter + 1;

(* Read motor status *)
Axis.ReadStatus();


(* Update states of Limit Switches *)
M_UpdateSwitches();

// 	Enable directions based on the state of STOP switches. 
//	Active LSTOP switch (stat.bStopSwitchNeg) disables motion in negative direction
//	Active USTOP switch (stat.bStopSwitchPos) disables motion in positive direction
Axis.PlcToNc.ControlDWord := AxisSetControllerEnable(Axis.PlcToNc.ControlDWord, stat.bEnabled);
Axis.PlcToNc.ControlDWord := AxisSetFeedEnableMinus(Axis.PlcToNc.ControlDWord, (NOT stat.bStopSwitchNeg));
Axis.PlcToNc.ControlDWord := AxisSetFeedEnablePlus(Axis.PlcToNc.ControlDWord,  (NOT stat.bStopSwitchPos));

(* 
	If both limit switches are active ((LSTOP & USTOP) or (LHW & UHW)), disable the motor and set error. 
	Do this check after NOVRAM configuration has been loaded. Doing it earlier
	could report some non-existing errors.
*)
IF	bNOVRAM_Loaded THEN
	IF 	stat.signals[E_MOTOR_SWITCH_INDEX.LSTOP].bActive AND stat.signals[E_MOTOR_SWITCH_INDEX.USTOP].bActive 	THEN
		stat.bEnabled 				:= FALSE;
		Axis.PlcToNc.ControlDWord 	:= AxisSetFeedEnableMinus(Axis.PlcToNc.ControlDWord, FALSE);
		Axis.PlcToNc.ControlDWord 	:= AxisSetFeedEnablePlus(Axis.PlcToNc.ControlDWord,  FALSE);
		M_SetError(E_MOTOR_ERROR.STOP_LIMITS_BOTH, 'ERROR: Both LSTOP and USTOP limits active. Motor disabled.');
	ELSIF 	stat.signals[E_MOTOR_SWITCH_INDEX.LHW].bActive AND stat.signals[E_MOTOR_SWITCH_INDEX.UHW].bActive 	THEN
		stat.bEnabled 				:= FALSE;
		Axis.PlcToNc.ControlDWord 	:= AxisSetFeedEnableMinus(Axis.PlcToNc.ControlDWord, FALSE);
		Axis.PlcToNc.ControlDWord 	:= AxisSetFeedEnablePlus(Axis.PlcToNc.ControlDWord,  FALSE);
		M_SetError(E_MOTOR_ERROR.HW_LIMITS_BOTH, 'ERROR: Both LHW and UHW limits active. Motor disabled.');
	END_IF
END_IF

(* Set velocity override to 100% *)
Axis.PlcToNc.Override := 1000000;


(* Check that Axis is in READY State *)
stat.bAxisReady := AxisIsReady(Axis.NcToPlc.StateDWord);

(* Read actual position and velocity. Circular optimised has normalised value *)
stat.lrPosActual	:= M_GetActualPos();
stat.lrVelActual	:= Axis.NcToPlc.ActVelo;
stat.lrPosError		:= Axis.NcToPlc.PosDiff;

(* Read Info data parameters *)
stat.nInfoData1	:= UINT_TO_INT(i_nInfoData1);
stat.nInfoData2	:= UINT_TO_INT(i_nInfoData2);

(* If brakes are not used, release them. Brakes are hard-coded to active low! *)
IF NOT cfg.bUseBrake THEN
	q_bBrake_Ctrl	:= M_GetLogicalState(state:= FALSE, activeLow:= TRUE);
END_IF

(* Get the state of the brake *)
stat.bBrakeActive	:= M_GetLogicalState(state:= i_bBrake_Stat, activeLow:= cfg.bActiveLowBrake);

// Get the In-Position status
stat.bInPosition	:= M_GetLogicalState(i_bInPos, cfg.bActiveLowInPos);

(* === Check for commands and internal events to be processed === *)
CheckForEvents();

(* === Process events according to the State Machine === *)
ProcessEvents();

METHOD ActionClearNOVRAM
VAR_INPUT
END_VAR
SetAction('ActionClearNOVRAM');

// Log event
M_LogEventStart('CLEAR NOVRAM');

M_NOVRAM_Clear(FALSE);		// Trigger M_NOVRAM_Clear()
END_METHOD

METHOD ActionErrExecute
VAR
END_VAR
SetAction('ActionErrExecute');

IF nEvent = E_MOTOR_EVENT.TIMEOUT_MOVE THEN
	M_SetStatus(E_MOTOR_ERROR.TIMEOUT_MOVE);
ELSIF nEvent = E_MOTOR_EVENT.TIMEOUT_SETPOS THEN
	M_SetStatus(E_MOTOR_ERROR.TIMEOUT_SETPOS);
END_IF
END_METHOD

METHOD ActionInitAbort
VAR_INPUT
END_VAR
SetAction('ActionInitAbort');

M_LogEventGeneral('Aborting INIT...');

// Set Error Status
M_SetStatus(E_MOTOR_ERROR.INIT_ABORTED);

// Release brakes. Brakes are hard-coded to active low!
q_bBrake_Ctrl	:= M_GetLogicalState(state:= FALSE, activeLow:= TRUE);


// Reset the timer for the command
toutCmd(IN:=FALSE);
toutCmd(IN:=TRUE,PT:=DINT_TO_TIME(cfg.nTimeoutInit));

// Restart HALT FB
fbHalt(Execute:=FALSE, Axis:=Axis);
//fbHalt(Execute:=TRUE, Axis:=Axis);

(*
IF NOT Axis.Status.NotMoving THEN
	// Restart the timer
	toutCmd(IN:=TRUE,PT:=DINT_TO_TIME(cfg.nTimeoutInit));
END_IF
*)

stat.bInitialised	:= FALSE;
//stat.bEnabled		:= FALSE;
stat.nInitStep		:= 0;
END_METHOD

METHOD ActionInitComplete
VAR_INPUT
END_VAR
SetAction('ActionInitComplete');

// Log event
M_LogEventEnd('INIT');

(* reply OK *)
stat.nErrorCode		:= E_MOTOR_ERROR.OK;
stat.sErrorText		:= 'OK';

(* Reset the timer action *)
toutCmd(IN:=FALSE);
END_METHOD

METHOD ActionInitExecute
VAR_INPUT
END_VAR
SetAction('ActionInitExecute');

// Log event
M_LogEventStart('INIT');

// Set starting states for all methods to be executed in INIT
nState_Init		:= MOTOR_INIT_STATE_RESET;
nState_Reset	:= MOTOR_RESET_STATE_START;
nState_InitSeq	:= MOTOR_INIT_SEQ_STATE_START;
nState_PreInit	:= MOTOR_PRE_INIT_STATE_START;
nState_PostInit	:= MOTOR_POST_INIT_STATE_START;

stat.bInitialised	:= FALSE;	// Clear the initialised flag

// Enable motor
stat.bEnabled	:= TRUE;

// Release brakes. Brakes are hard-coded to active low!
q_bBrake_Ctrl	:= M_GetLogicalState(state:= FALSE, activeLow:= TRUE);

// Start the cmd timer.
// Give 5 sec more than the timeout for INIT sequence
toutCmd(IN:=FALSE);
toutCmd(IN:=TRUE,PT:=DINT_TO_TIME(cfg.nTimeoutInit+5000));
END_METHOD

METHOD ActionInitReject
VAR_INPUT
END_VAR
SetAction('ActionInitReject');

(* Reject an INIT command since another one is in progress. *)
(* do not reset the timer ... *)
END_METHOD

METHOD ActionMoveExecute
VAR_INPUT
END_VAR
SetAction('ActionMoveExecute');

(* Clear the error *)
M_SetStatus(E_MOTOR_ERROR.OK);

(* 
	MOVE RELATIVE is converted to MOVE ABSOLUTE
	We just add the offset to the current position and move absolute!
*)
IF ctrl.nMoveType = E_MOTOR_MOVE_TYPE.RELATIVE THEN
	M_LogEventMoveRel(ctrl.lrOffset, stat.lrPosActual, ctrl.lrVelocity);
	M_LogEventDebug('MOVEREL converted to MOVEABS');
	ctrl.lrPosition		:= stat.lrPosActual + ctrl.lrOffset;	(* Set new absolute position *)
	ctrl.nMoveType 		:= E_MOTOR_MOVE_TYPE.ABSOLUTE; 
END_IF


// Handling of Locked function. 
// If the motor is locked, there is no need to prepare anything here.
// We just exit this method.
// Method ActivityMoving() will do a check and set error, if needed.
IF 	cfg.bLock THEN
	// Nothing to do - exit this method.
	RETURN;
END_IF


